LIN {X 0,Y 485.77,Z 296.531,A -85,B 0,C 180,E1 -14643.447,E2 -14643.447} C_VEL
LIN {X 0,Y 485.784,Z 296.534,A -85,B 0,C 180,E1 -14646.187,E2 -14646.187} C_VEL
LIN {X 0,Y 485.815,Z 296.524,A -85,B 0,C 180,E1 -14648.87,E2 -14648.87} C_VEL
LIN {X 0,Y 485.863,Z 296.525,A -85,B 0,C 180,E1 -14652.08,E2 -14652.08} C_VEL
LIN {X 0,Y 485.883,Z 296.515,A -85,B 0,C 180,E1 -14654.987,E2 -14654.987} C_VEL
LIN {X 0,Y 485.919,Z 296.513,A -85,B 0,C 180,E1 -14658.355,E2 -14658.355} C_VEL
LIN {X 0,Y 485.937,Z 296.624,A -85,B 0,C 180,E1 -14661.371,E2 -14661.371} C_VEL
LIN {X 0,Y 487.362,Z 304.386,A -85,B 0,C 180,E1 -14663.005,E2 -14663.005} C_VEL
LIN {X 0,Y 489.641,Z 313.003,A -85,B 0,C 180,E1 -14663.215,E2 -14663.215} C_VEL
LIN {X 0,Y 492.442,Z 326.863,A -85,B 0,C 180,E1 -14663.515,E2 -14663.515} C_VEL
LIN {X 0,Y 490.89,Z 439.426,A -85,B 0,C 180,E1 -14665.164,E2 -14665.164} C_VEL
LIN {X 0,Y 490.643,Z 451.445,A -85,B 0,C 180,E1 -14665.464,E2 -14665.464} C_VEL
LIN {X 0,Y 489.693,Z 457.148,A -85,B 0,C 180,E1 -14665.617,E2 -14665.617} C_VEL
LIN {X 0,Y 486.571,Z 466.299,A -85,B 0,C 180,E1 -14665.884,E2 -14665.884} C_VEL
LIN {X 0,Y 483.496,Z 475.212,A -85,B 0,C 180,E1 -14666.236,E2 -14666.236} C_VEL
LIN {X 0,Y 482.618,Z 480.534,A -85,B 0,C 180,E1 -14666.517,E2 -14666.517} C_VEL
LIN {X 0,Y 481.935,Z 493.871,A -85,B 0,C 180,E1 -14667.395,E2 -14667.395} C_VEL
LIN {X 0,Y 480.98,Z 505.372,A -85,B 0,C 180,E1 -14668.329,E2 -14668.329} C_VEL
LIN {X 0,Y 480.395,Z 515.838,A -85,B 0,C 180,E1 -14669.371,E2 -14669.371} C_VEL
LIN {X 0,Y 479.518,Z 526.296,A -85,B 0,C 180,E1 -14670.626,E2 -14670.626} C_VEL
LIN {X 0,Y 478.886,Z 534.915,A -85,B 0,C 180,E1 -14671.884,E2 -14671.884} C_VEL
LIN {X 0,Y 478.287,Z 542.104,A -85,B 0,C 180,E1 -14673.146,E2 -14673.146} C_VEL
LIN {X 0,Y 477.979,Z 549.726,A -85,B 0,C 180,E1 -14674.801,E2 -14674.801} C_VEL
LIN {X 0,Y 477.604,Z 555.152,A -85,B 0,C 180,E1 -14676.313,E2 -14676.313} C_VEL
LIN {X 0,Y 477.361,Z 558.684,A -85,B 0,C 180,E1 -14677.586,E2 -14677.586} C_VEL
LIN {X 0,Y 477.178,Z 562.146,A -85,B 0,C 180,E1 -14679.29,E2 -14679.29} C_VEL
LIN {X 0,Y 477.117,Z 564.216,A -85,B 0,C 180,E1 -14681,E2 -14681} C_VEL
LIN {X 0,Y 477.101,Z 564.93,A -85,B 0,C 180,E1 -14682.72,E2 -14682.72} C_VEL
LIN {X 0,Y 477.337,Z 564.263,A -85,B 0,C 180,E1 -14684.443,E2 -14684.443} C_VEL
LIN {X 0,Y 477.485,Z 562.216,A -85,B 0,C 180,E1 -14686.181,E2 -14686.181} C_VEL
LIN {X 0,Y 477.942,Z 558.707,A -85,B 0,C 180,E1 -14687.922,E2 -14687.922} C_VEL
LIN {X 0,Y 478.56,Z 553.62,A -85,B 0,C 180,E1 -14689.67,E2 -14689.67} C_VEL
LIN {X 0,Y 479.118,Z 548.633,A -85,B 0,C 180,E1 -14690.985,E2 -14690.985} C_VEL
LIN {X 0,Y 480.003,Z 541.388,A -85,B 0,C 180,E1 -14692.52,E2 -14692.52} C_VEL
LIN {X 0,Y 480.959,Z 533.698,A -85,B 0,C 180,E1 -14693.839,E2 -14693.839} C_VEL
LIN {X 0,Y 482.026,Z 524.437,A -85,B 0,C 180,E1 -14695.15,E2 -14695.15} C_VEL
LIN {X 0,Y 483.19,Z 514.097,A -85,B 0,C 180,E1 -14696.353,E2 -14696.353} C_VEL
LIN {X 0,Y 484.363,Z 502.622,A -85,B 0,C 180,E1 -14697.446,E2 -14697.446} C_VEL
LIN {X 0,Y 485.333,Z 491.49,A -85,B 0,C 180,E1 -14698.313,E2 -14698.313} C_VEL
LIN {X 0,Y 486.333,Z 478.223,A -85,B 0,C 180,E1 -14699.14,E2 -14699.14} C_VEL
LIN {X 0,Y 487.079,Z 464.484,A -85,B 0,C 180,E1 -14699.801,E2 -14699.801} C_VEL
LIN {X 0,Y 487.718,Z 449.719,A -85,B 0,C 180,E1 -14700.31,E2 -14700.31} C_VEL
LIN {X 0,Y 488.109,Z 435.76,A -85,B 0,C 180,E1 -14700.619,E2 -14700.619} C_VEL
LIN {X 0,Y 489.875,Z 330.426,A -85,B 0,C 180,E1 -14702.194,E2 -14702.194} C_VEL
LIN {X 0,Y 488.073,Z 324.325,A -85,B 0,C 180,E1 -14702.385,E2 -14702.385} C_VEL
LIN {X 0,Y 480.502,Z 305.747,A -85,B 0,C 180,E1 -14703.112,E2 -14703.112} C_VEL
LIN {X 0,Y 478.693,Z 297.414,A -85,B 0,C 180,E1 -14705.071,E2 -14705.071} C_VEL
LIN {X 0,Y 478.681,Z 297.417,A -85,B 0,C 180,E1 -14707.918,E2 -14707.918} C_VEL
LIN {X 0,Y 478.695,Z 297.409,A -85,B 0,C 180,E1 -14711.179,E2 -14711.179} C_VEL
LIN {X 0,Y 478.716,Z 297.403,A -85,B 0,C 180,E1 -14714.196,E2 -14714.196} C_VEL
LIN {X 0,Y 478.703,Z 297.412,A -85,B 0,C 180,E1 -14717.017,E2 -14717.017} C_VEL
LIN {X 0,Y 478.708,Z 297.412,A -85,B 0,C 180,E1 -14719.924,E2 -14719.924} C_VEL
LIN {X 0,Y 478.721,Z 297.402,A -85,B 0,C 180,E1 -14723.138,E2 -14723.138} C_VEL
LIN {X 0,Y 478.69,Z 297.412,A -85,B 0,C 180,E1 -14726.218,E2 -14726.218} C_VEL
LIN {X 0,Y 478.703,Z 297.407,A -85,B 0,C 180,E1 -14729.195,E2 -14729.195} C_VEL
LIN {X 0,Y 478.741,Z 297.401,A -85,B 0,C 180,E1 -14732.083,E2 -14732.083} C_VEL
LIN {X 0,Y 478.725,Z 297.41,A -85,B 0,C 180,E1 -14735.108,E2 -14735.108} C_VEL
LIN {X 0,Y 478.751,Z 297.404,A -85,B 0,C 180,E1 -14738.545,E2 -14738.545} C_VEL
LIN {X 0,Y 478.762,Z 297.398,A -85,B 0,C 180,E1 -14741.224,E2 -14741.224} C_VEL
LIN {X 0,Y 478.812,Z 297.397,A -85,B 0,C 180,E1 -14744.895,E2 -14744.895} C_VEL
LIN {X 0,Y 478.849,Z 297.392,A -85,B 0,C 180,E1 -14748.183,E2 -14748.183} C_VEL
LIN {X 0,Y 478.887,Z 297.383,A -85,B 0,C 180,E1 -14751.589,E2 -14751.589} C_VEL
LIN {X 0,Y 478.991,Z 297.376,A -85,B 0,C 180,E1 -14754.966,E2 -14754.966} C_VEL
LIN {X 0,Y 478.798,Z 297.397,A -85,B 0,C 180,E1 -14757.485,E2 -14757.485} C_VEL
LIN {X 0,Y 479.032,Z 297.368,A -85,B 0,C 180,E1 -14760,E2 -14760} C_VEL
LIN {X 0,Y 478.98,Z 297.375,A -85,B 0,C 180,E1 -14764.193,E2 -14764.193} C_VEL
LIN {X 0,Y 478.917,Z 297.378,A -85,B 0,C 180,E1 -14766.719,E2 -14766.719} C_VEL
LIN {X 0,Y 478.863,Z 297.392,A -85,B 0,C 180,E1 -14769.259,E2 -14769.259} C_VEL
LIN {X 0,Y 478.898,Z 297.377,A -85,B 0,C 180,E1 -14771.816,E2 -14771.816} C_VEL
LIN {X 0,Y 478.856,Z 297.39,A -85,B 0,C 180,E1 -14775.266,E2 -14775.266} C_VEL
LIN {X 0,Y 478.778,Z 297.398,A -85,B 0,C 180,E1 -14778.775,E2 -14778.775} C_VEL
LIN {X 0,Y 478.751,Z 297.397,A -85,B 0,C 180,E1 -14781.455,E2 -14781.455} C_VEL
LIN {X 0,Y 478.725,Z 297.409,A -85,B 0,C 180,E1 -14784.892,E2 -14784.892} C_VEL
LIN {X 0,Y 478.741,Z 297.405,A -85,B 0,C 180,E1 -14787.917,E2 -14787.917} C_VEL
LIN {X 0,Y 478.725,Z 297.407,A -85,B 0,C 180,E1 -14790.804,E2 -14790.804} C_VEL
LIN {X 0,Y 478.741,Z 297.404,A -85,B 0,C 180,E1 -14793.778,E2 -14793.778} C_VEL
LIN {X 0,Y 478.784,Z 297.387,A -85,B 0,C 180,E1 -14796.857,E2 -14796.857} C_VEL
LIN {X 0,Y 478.754,Z 297.405,A -85,B 0,C 180,E1 -14800.072,E2 -14800.072} C_VEL
LIN {X 0,Y 478.732,Z 297.406,A -85,B 0,C 180,E1 -14803.446,E2 -14803.446} C_VEL
LIN {X 0,Y 478.719,Z 297.411,A -85,B 0,C 180,E1 -14806.556,E2 -14806.556} C_VEL
LIN {X 0,Y 478.747,Z 297.406,A -85,B 0,C 180,E1 -14809.535,E2 -14809.535} C_VEL
LIN {X 0,Y 478.781,Z 297.408,A -85,B 0,C 180,E1 -14812.186,E2 -14812.186} C_VEL
LIN {X 0,Y 478.744,Z 297.414,A -85,B 0,C 180,E1 -14815.211,E2 -14815.211} C_VEL
LIN {X 0,Y 478.763,Z 297.414,A -85,B 0,C 180,E1 -14818.221,E2 -14818.221} C_VEL
LIN {X 0,Y 478.75,Z 297.508,A -85,B 0,C 180,E1 -14819.048,E2 -14819.048} C_VEL
LIN {X 0,Y 482.247,Z 312.121,A -85,B 0,C 180,E1 -14821.836,E2 -14821.836} C_VEL
LIN {X 0,Y 484.81,Z 324.657,A -85,B 0,C 180,E1 -14824.101,E2 -14824.101} C_VEL
LIN {X 0,Y 483.591,Z 338.406,A -85,B 0,C 180,E1 -14826.303,E2 -14826.303} C_VEL
LIN {X 0,Y 481.96,Z 355.754,A -85,B 0,C 180,E1 -14829.033,E2 -14829.033} C_VEL
LIN {X 0,Y 486.987,Z 384.746,A -85,B 0,C 180,E1 -14829.76,E2 -14829.76} C_VEL
LIN {X 0,Y 488.865,Z 398.674,A -85,B 0,C 180,E1 -14830.074,E2 -14830.074} C_VEL
LIN {X 0,Y 487.289,Z 493.967,A -85,B 0,C 180,E1 -14831.513,E2 -14831.513} C_VEL
LIN {X 0,Y 486.53,Z 508.818,A -85,B 0,C 180,E1 -14831.899,E2 -14831.899} C_VEL
LIN {X 0,Y 485.571,Z 522.508,A -85,B 0,C 180,E1 -14832.423,E2 -14832.423} C_VEL
LIN {X 0,Y 484.462,Z 535.489,A -85,B 0,C 180,E1 -14833.086,E2 -14833.086} C_VEL
LIN {X 0,Y 483.26,Z 548.083,A -85,B 0,C 180,E1 -14833.909,E2 -14833.909} C_VEL
LIN {X 0,Y 481.995,Z 559.586,A -85,B 0,C 180,E1 -14834.839,E2 -14834.839} C_VEL
LIN {X 0,Y 480.873,Z 570.17,A -85,B 0,C 180,E1 -14835.881,E2 -14835.881} C_VEL
LIN {X 0,Y 479.709,Z 580.705,A -85,B 0,C 180,E1 -14837.136,E2 -14837.136} C_VEL
LIN {X 0,Y 478.789,Z 590.546,A -85,B 0,C 180,E1 -14838.573,E2 -14838.573} C_VEL
LIN {X 0,Y 477.939,Z 598.91,A -85,B 0,C 180,E1 -14840.086,E2 -14840.086} C_VEL
LIN {X 0,Y 477.375,Z 605.499,A -85,B 0,C 180,E1 -14841.565,E2 -14841.565} C_VEL
LIN {X 0,Y 476.995,Z 617.328,A -85,B 0,C 180,E1 -14844.947,E2 -14844.947} C_VEL
LIN {X 0,Y 476.94,Z 621.761,A -85,B 0,C 180,E1 -14846.634,E2 -14846.634} C_VEL
LIN {X 0,Y 476.957,Z 624.638,A -85,B 0,C 180,E1 -14848.319,E2 -14848.319} C_VEL
LIN {X 0,Y 477.003,Z 625.52,A -85,B 0,C 180,E1 -14849.161,E2 -14849.161} C_VEL
LIN {X 0,Y 476.959,Z 626.175,A -85,B 0,C 180,E1 -14850.843,E2 -14850.843} C_VEL
LIN {X 0,Y 476.924,Z 625.353,A -85,B 0,C 180,E1 -14852.527,E2 -14852.527} C_VEL
LIN {X 0,Y 476.963,Z 623.088,A -85,B 0,C 180,E1 -14854.213,E2 -14854.213} C_VEL
LIN {X 0,Y 477.08,Z 619.333,A -85,B 0,C 180,E1 -14855.901,E2 -14855.901} C_VEL
LIN {X 0,Y 477.383,Z 614.001,A -85,B 0,C 180,E1 -14857.59,E2 -14857.59} C_VEL
LIN {X 0,Y 477.739,Z 608.828,A -85,B 0,C 180,E1 -14858.858,E2 -14858.858} C_VEL
LIN {X 0,Y 478.476,Z 601.406,A -85,B 0,C 180,E1 -14860.333,E2 -14860.333} C_VEL
LIN {X 0,Y 479.204,Z 593.155,A -85,B 0,C 180,E1 -14861.67,E2 -14861.67} C_VEL
LIN {X 0,Y 480.028,Z 584.334,A -85,B 0,C 180,E1 -14862.859,E2 -14862.859} C_VEL
LIN {X 0,Y 480.975,Z 574.091,A -85,B 0,C 180,E1 -14864.013,E2 -14864.013} C_VEL
LIN {X 0,Y 482.133,Z 562.839,A -85,B 0,C 180,E1 -14865.053,E2 -14865.053} C_VEL
LIN {X 0,Y 483.157,Z 550.55,A -85,B 0,C 180,E1 -14865.991,E2 -14865.991} C_VEL
LIN {X 0,Y 484.352,Z 536.947,A -85,B 0,C 180,E1 -14866.814,E2 -14866.814} C_VEL
LIN {X 0,Y 485.362,Z 522.74,A -85,B 0,C 180,E1 -14867.481,E2 -14867.481} C_VEL
LIN {X 0,Y 486.254,Z 508.664,A -85,B 0,C 180,E1 -14867.959,E2 -14867.959} C_VEL
LIN {X 0,Y 486.975,Z 491.209,A -85,B 0,C 180,E1 -14868.346,E2 -14868.346} C_VEL
LIN {X 0,Y 489.953,Z 399.064,A -85,B 0,C 180,E1 -14870.171,E2 -14870.171} C_VEL
LIN {X 0,Y 488.283,Z 381.463,A -85,B 0,C 180,E1 -14870.68,E2 -14870.68} C_VEL
LIN {X 0,Y 484.759,Z 358.037,A -85,B 0,C 180,E1 -14871.468,E2 -14871.468} C_VEL
LIN {X 0,Y 483.933,Z 352.73,A -85,B 0,C 180,E1 -14871.699,E2 -14871.699} C_VEL
LIN {X 0,Y 481.685,Z 333.484,A -85,B 0,C 180,E1 -14872.865,E2 -14872.865} C_VEL
LIN {X 0,Y 482.771,Z 318.818,A -85,B 0,C 180,E1 -14875.113,E2 -14875.113} C_VEL
LIN {X 0,Y 480.649,Z 306.868,A -85,B 0,C 180,E1 -14877.094,E2 -14877.094} C_VEL
LIN {X 0,Y 478.775,Z 297.404,A -85,B 0,C 180,E1 -14878.705,E2 -14878.705} C_VEL
LIN {X 0,Y 478.675,Z 297.414,A -85,B 0,C 180,E1 -14881.928,E2 -14881.928} C_VEL
LIN {X 0,Y 478.711,Z 297.414,A -85,B 0,C 180,E1 -14884.977,E2 -14884.977} C_VEL
LIN {X 0,Y 478.676,Z 297.417,A -85,B 0,C 180,E1 -14887.924,E2 -14887.924} C_VEL
LIN {X 0,Y 478.708,Z 297.412,A -85,B 0,C 180,E1 -14890.46,E2 -14890.46} C_VEL
LIN {X 0,Y 478.739,Z 297.408,A -85,B 0,C 180,E1 -14893.447,E2 -14893.447} C_VEL
LIN {X 0,Y 478.74,Z 297.409,A -85,B 0,C 180,E1 -14896.555,E2 -14896.555} C_VEL
LIN {X 0,Y 478.708,Z 297.411,A -85,B 0,C 180,E1 -14899.542,E2 -14899.542} C_VEL
LIN {X 0,Y 478.71,Z 297.413,A -85,B 0,C 180,E1 -14902.199,E2 -14902.199} C_VEL
LIN {X 0,Y 478.747,Z 297.408,A -85,B 0,C 180,E1 -14905.208,E2 -14905.208} C_VEL
LIN {X 0,Y 478.718,Z 297.413,A -85,B 0,C 180,E1 -14908.214,E2 -14908.214} C_VEL
LIN {X 0,Y 478.757,Z 297.405,A -85,B 0,C 180,E1 -14911.384,E2 -14911.384} C_VEL
LIN {X 0,Y 478.733,Z 297.412,A -85,B 0,C 180,E1 -14913.964,E2 -14913.964} C_VEL
LIN {X 0,Y 478.761,Z 297.411,A -85,B 0,C 180,E1 -14917.181,E2 -14917.181} C_VEL
LIN {X 0,Y 478.785,Z 297.414,A -85,B 0,C 180,E1 -14920.337,E2 -14920.337} C_VEL
LIN {X 0,Y 478.83,Z 297.543,A -85,B 0,C 180,E1 -14922.632,E2 -14922.632} C_VEL
LIN {X 0,Y 483.17,Z 311.983,A -85,B 0,C 180,E1 -14925.304,E2 -14925.304} C_VEL
LIN {X 0,Y 486.011,Z 325.005,A -85,B 0,C 180,E1 -14927.515,E2 -14927.515} C_VEL
LIN {X 0,Y 486.185,Z 329.106,A -85,B 0,C 180,E1 -14928.153,E2 -14928.153} C_VEL
LIN {X 0,Y 485.162,Z 345.213,A -85,B 0,C 180,E1 -14930.495,E2 -14930.495} C_VEL
LIN {X 0,Y 490.051,Z 367.792,A -85,B 0,C 180,E1 -14931.354,E2 -14931.354} C_VEL
LIN {X 0,Y 491.129,Z 374.172,A -85,B 0,C 180,E1 -14931.568,E2 -14931.568} C_VEL
LIN {X 0,Y 487.703,Z 474.381,A -85,B 0,C 180,E1 -14933.532,E2 -14933.532} C_VEL
LIN {X 0,Y 487.049,Z 490.57,A -85,B 0,C 180,E1 -14933.912,E2 -14933.912} C_VEL
LIN {X 0,Y 486.356,Z 504.272,A -85,B 0,C 180,E1 -14934.396,E2 -14934.396} C_VEL
LIN {X 0,Y 485.275,Z 518.802,A -85,B 0,C 180,E1 -14935.083,E2 -14935.083} C_VEL
LIN {X 0,Y 484.276,Z 531.323,A -85,B 0,C 180,E1 -14935.853,E2 -14935.853} C_VEL
LIN {X 0,Y 483.13,Z 543.526,A -85,B 0,C 180,E1 -14936.779,E2 -14936.779} C_VEL
LIN {X 0,Y 482.019,Z 555.678,A -85,B 0,C 180,E1 -14937.918,E2 -14937.918} C_VEL
LIN {X 0,Y 480.878,Z 566.583,A -85,B 0,C 180,E1 -14939.165,E2 -14939.165} C_VEL
LIN {X 0,Y 479.753,Z 575.623,A -85,B 0,C 180,E1 -14940.418,E2 -14940.418} C_VEL
LIN {X 0,Y 478.88,Z 584.231,A -85,B 0,C 180,E1 -14941.886,E2 -14941.886} C_VEL
LIN {X 0,Y 478.087,Z 591.225,A -85,B 0,C 180,E1 -14943.36,E2 -14943.36} C_VEL
LIN {X 0,Y 477.836,Z 595.873,A -85,B 0,C 180,E1 -14944.579,E2 -14944.579} C_VEL
LIN {X 0,Y 477.453,Z 599.934,A -85,B 0,C 180,E1 -14945.894,E2 -14945.894} C_VEL
LIN {X 0,Y 477.069,Z 603.711,A -85,B 0,C 180,E1 -14947.593,E2 -14947.593} C_VEL
LIN {X 0,Y 476.906,Z 606.01,A -85,B 0,C 180,E1 -14949.297,E2 -14949.297} C_VEL
LIN {X 0,Y 476.914,Z 606.669,A -85,B 0,C 180,E1 -14950.247,E2 -14950.247} C_VEL
LIN {X 0,Y 476.739,Z 606.749,A -85,B 0,C 180,E1 -14951.87,E2 -14951.87} C_VEL
LIN {X 0,Y 476.784,Z 605.387,A -85,B 0,C 180,E1 -14953.595,E2 -14953.595} C_VEL
LIN {X 0,Y 476.834,Z 604.117,A -85,B 0,C 180,E1 -14954.461,E2 -14954.461} C_VEL
LIN {X 0,Y 476.931,Z 600.386,A -85,B 0,C 180,E1 -14956.203,E2 -14956.203} C_VEL
LIN {X 0,Y 477.083,Z 596.142,A -85,B 0,C 180,E1 -14957.614,E2 -14957.614} C_VEL
LIN {X 0,Y 477.386,Z 589.572,A -85,B 0,C 180,E1 -14959.277,E2 -14959.277} C_VEL
LIN {X 0,Y 477.755,Z 581.739,A -85,B 0,C 180,E1 -14960.826,E2 -14960.826} C_VEL
LIN {X 0,Y 478.214,Z 573.386,A -85,B 0,C 180,E1 -14962.158,E2 -14962.158} C_VEL
LIN {X 0,Y 478.832,Z 563.194,A -85,B 0,C 180,E1 -14963.492,E2 -14963.492} C_VEL
LIN {X 0,Y 479.486,Z 551.781,A -85,B 0,C 180,E1 -14964.719,E2 -14964.719} C_VEL
LIN {X 0,Y 480.154,Z 540.357,A -85,B 0,C 180,E1 -14965.727,E2 -14965.727} C_VEL
LIN {X 0,Y 480.828,Z 528.102,A -85,B 0,C 180,E1 -14966.612,E2 -14966.612} C_VEL
LIN {X 0,Y 481.466,Z 514.839,A -85,B 0,C 180,E1 -14967.377,E2 -14967.377} C_VEL
LIN {X 0,Y 482.085,Z 500.781,A -85,B 0,C 180,E1 -14968.001,E2 -14968.001} C_VEL
LIN {X 0,Y 482.647,Z 486.247,A -85,B 0,C 180,E1 -14968.467,E2 -14968.467} C_VEL
LIN {X 0,Y 483.012,Z 468.488,A -85,B 0,C 180,E1 -14968.828,E2 -14968.828} C_VEL
LIN {X 0,Y 484.847,Z 370.517,A -85,B 0,C 180,E1 -14970.589,E2 -14970.589} C_VEL
LIN {X 0,Y 481.086,Z 343.578,A -85,B 0,C 180,E1 -14971.22,E2 -14971.22} C_VEL
LIN {X 0,Y 481.95,Z 323.747,A -85,B 0,C 180,E1 -14974.062,E2 -14974.062} C_VEL
LIN {X 0,Y 482.272,Z 315.444,A -85,B 0,C 180,E1 -14975.255,E2 -14975.255} C_VEL
LIN {X 0,Y 479,Z 298.562,A -85,B 0,C 180,E1 -14977.846,E2 -14977.846} C_VEL
LIN {X 0,Y 478.724,Z 297.412,A -85,B 0,C 180,E1 -14978.05,E2 -14978.05} C_VEL
LIN {X 0,Y 478.719,Z 297.408,A -85,B 0,C 180,E1 -14981.18,E2 -14981.18} C_VEL
LIN {X 0,Y 478.739,Z 297.411,A -85,B 0,C 180,E1 -14984.197,E2 -14984.197} C_VEL
LIN {X 0,Y 478.714,Z 297.409,A -85,B 0,C 180,E1 -14987.02,E2 -14987.02} C_VEL
LIN {X 0,Y 478.696,Z 297.414,A -85,B 0,C 180,E1 -14989.921,E2 -14989.921} C_VEL
LIN {X 0,Y 478.674,Z 297.414,A -85,B 0,C 180,E1 -14993.132,E2 -14993.132} C_VEL
LIN {X 0,Y 478.701,Z 297.416,A -85,B 0,C 180,E1 -14996.217,E2 -14996.217} C_VEL
LIN {X 0,Y 478.723,Z 297.41,A -85,B 0,C 180,E1 -14999.685,E2 -14999.685} C_VEL
LIN {X 0,Y 478.743,Z 297.411,A -85,B 0,C 180,E1 -15002.081,E2 -15002.081} C_VEL
LIN {X 0,Y 478.752,Z 297.404,A -85,B 0,C 180,E1 -15005.108,E2 -15005.108} C_VEL
LIN {X 0,Y 478.78,Z 297.402,A -85,B 0,C 180,E1 -15008.545,E2 -15008.545} C_VEL
LIN {X 0,Y 478.824,Z 297.401,A -85,B 0,C 180,E1 -15011.961,E2 -15011.961} C_VEL
LIN {X 0,Y 478.843,Z 297.392,A -85,B 0,C 180,E1 -15014.892,E2 -15014.892} C_VEL
LIN {X 0,Y 478.876,Z 297.392,A -85,B 0,C 180,E1 -15018.182,E2 -15018.182} C_VEL
LIN {X 0,Y 478.9,Z 297.528,A -85,B 0,C 180,E1 -15021.217,E2 -15021.217} C_VEL
LIN {X 0,Y 480.268,Z 304.765,A -85,B 0,C 180,E1 -15022.76,E2 -15022.76} C_VEL
LIN {X 0,Y 482.973,Z 314.716,A -85,B 0,C 180,E1 -15023.016,E2 -15023.016} C_VEL
LIN {X 0,Y 485.65,Z 329.013,A -85,B 0,C 180,E1 -15023.323,E2 -15023.323} C_VEL
LIN {X 0,Y 484.007,Z 439.783,A -85,B 0,C 180,E1 -15024.965,E2 -15024.965} C_VEL
LIN {X 0,Y 483.662,Z 454.476,A -85,B 0,C 180,E1 -15025.351,E2 -15025.351} C_VEL
LIN {X 0,Y 483.145,Z 468.419,A -85,B 0,C 180,E1 -15025.893,E2 -15025.893} C_VEL
LIN {X 0,Y 482.618,Z 480.534,A -85,B 0,C 180,E1 -15026.517,E2 -15026.517} C_VEL
LIN {X 0,Y 481.676,Z 485.877,A -85,B 0,C 180,E1 -15026.822,E2 -15026.822} C_VEL
LIN {X 0,Y 478.298,Z 494.251,A -85,B 0,C 180,E1 -15027.321,E2 -15027.321} C_VEL
LIN {X 0,Y 474.914,Z 502.288,A -85,B 0,C 180,E1 -15027.879,E2 -15027.879} C_VEL
LIN {X 0,Y 473.928,Z 506.979,A -85,B 0,C 180,E1 -15028.284,E2 -15028.284} C_VEL
LIN {X 0,Y 473.357,Z 517.422,A -85,B 0,C 180,E1 -15029.362,E2 -15029.362} C_VEL
LIN {X 0,Y 472.427,Z 527.691,A -85,B 0,C 180,E1 -15030.635,E2 -15030.635} C_VEL
LIN {X 0,Y 471.824,Z 536.145,A -85,B 0,C 180,E1 -15031.912,E2 -15031.912} C_VEL
LIN {X 0,Y 471.114,Z 544.258,A -85,B 0,C 180,E1 -15033.407,E2 -15033.407} C_VEL
LIN {X 0,Y 470.913,Z 550.161,A -85,B 0,C 180,E1 -15034.746,E2 -15034.746} C_VEL
LIN {X 0,Y 470.499,Z 555.958,A -85,B 0,C 180,E1 -15036.409,E2 -15036.409} C_VEL
LIN {X 0,Y 470.245,Z 559.431,A -85,B 0,C 180,E1 -15037.702,E2 -15037.702} C_VEL
LIN {X 0,Y 470.084,Z 562.787,A -85,B 0,C 180,E1 -15039.431,E2 -15039.431} C_VEL
LIN {X 0,Y 470.029,Z 564.736,A -85,B 0,C 180,E1 -15041.168,E2 -15041.168} C_VEL
LIN {X 0,Y 470.034,Z 565.327,A -85,B 0,C 180,E1 -15042.914,E2 -15042.914} C_VEL
LIN {X 0,Y 470.265,Z 564.557,A -85,B 0,C 180,E1 -15044.665,E2 -15044.665} C_VEL
LIN {X 0,Y 470.457,Z 562.408,A -85,B 0,C 180,E1 -15046.43,E2 -15046.43} C_VEL
LIN {X 0,Y 470.959,Z 558.794,A -85,B 0,C 180,E1 -15048.197,E2 -15048.197} C_VEL
LIN {X 0,Y 471.637,Z 553.596,A -85,B 0,C 180,E1 -15049.971,E2 -15049.971} C_VEL
LIN {X 0,Y 472.229,Z 548.487,A -85,B 0,C 180,E1 -15051.307,E2 -15051.307} C_VEL
LIN {X 0,Y 473.183,Z 541.11,A -85,B 0,C 180,E1 -15052.863,E2 -15052.863} C_VEL
LIN {X 0,Y 474.19,Z 533.298,A -85,B 0,C 180,E1 -15054.196,E2 -15054.196} C_VEL
LIN {X 0,Y 475.335,Z 523.936,A -85,B 0,C 180,E1 -15055.516,E2 -15055.516} C_VEL
LIN {X 0,Y 476.56,Z 513.234,A -85,B 0,C 180,E1 -15056.749,E2 -15056.749} C_VEL
LIN {X 0,Y 477.822,Z 501.422,A -85,B 0,C 180,E1 -15057.854,E2 -15057.854} C_VEL
LIN {X 0,Y 478.829,Z 490.016,A -85,B 0,C 180,E1 -15058.727,E2 -15058.727} C_VEL
LIN {X 0,Y 479.822,Z 477.164,A -85,B 0,C 180,E1 -15059.514,E2 -15059.514} C_VEL
LIN {X 0,Y 480.516,Z 464.313,A -85,B 0,C 180,E1 -15060.129,E2 -15060.129} C_VEL
LIN {X 0,Y 481.157,Z 449.886,A -85,B 0,C 180,E1 -15060.628,E2 -15060.628} C_VEL
LIN {X 0,Y 481.555,Z 436.381,A -85,B 0,C 180,E1 -15060.93,E2 -15060.93} C_VEL
LIN {X 0,Y 483.353,Z 331.59,A -85,B 0,C 180,E1 -15062.519,E2 -15062.519} C_VEL
LIN {X 0,Y 481.848,Z 326.725,A -85,B 0,C 180,E1 -15062.679,E2 -15062.679} C_VEL
LIN {X 0,Y 474.63,Z 309.241,A -85,B 0,C 180,E1 -15063.368,E2 -15063.368} C_VEL
LIN {X 0,Y 473.384,Z 306.242,A -85,B 0,C 180,E1 -15063.503,E2 -15063.503} C_VEL
LIN {X 0,Y 471.633,Z 298.296,A -85,B 0,C 180,E1 -15065.424,E2 -15065.424} C_VEL
LIN {X 0,Y 471.621,Z 298.29,A -85,B 0,C 180,E1 -15068.589,E2 -15068.589} C_VEL
LIN {X 0,Y 471.653,Z 298.286,A -85,B 0,C 180,E1 -15071.931,E2 -15071.931} C_VEL
LIN {X 0,Y 471.69,Z 298.274,A -85,B 0,C 180,E1 -15074.538,E2 -15074.538} C_VEL
LIN {X 0,Y 471.653,Z 298.291,A -85,B 0,C 180,E1 -15077.944,E2 -15077.944} C_VEL
LIN {X 0,Y 471.671,Z 298.288,A -85,B 0,C 180,E1 -15080.549,E2 -15080.549} C_VEL
LIN {X 0,Y 471.685,Z 298.27,A -85,B 0,C 180,E1 -15083.559,E2 -15083.559} C_VEL
LIN {X 0,Y 471.639,Z 298.29,A -85,B 0,C 180,E1 -15086.667,E2 -15086.667} C_VEL
LIN {X 0,Y 471.679,Z 298.285,A -85,B 0,C 180,E1 -15089.675,E2 -15089.675} C_VEL
LIN {X 0,Y 471.704,Z 298.275,A -85,B 0,C 180,E1 -15092.987,E2 -15092.987} C_VEL
LIN {X 0,Y 471.666,Z 298.291,A -85,B 0,C 180,E1 -15095.43,E2 -15095.43} C_VEL
LIN {X 0,Y 471.708,Z 298.283,A -85,B 0,C 180,E1 -15098.209,E2 -15098.209} C_VEL
LIN {X 0,Y 471.704,Z 298.277,A -85,B 0,C 180,E1 -15100.932,E2 -15100.932} C_VEL
LIN {X 0,Y 471.736,Z 298.277,A -85,B 0,C 180,E1 -15104.498,E2 -15104.498} C_VEL
LIN {X 0,Y 471.768,Z 298.27,A -85,B 0,C 180,E1 -15107.132,E2 -15107.132} C_VEL
LIN {X 0,Y 471.785,Z 298.268,A -85,B 0,C 180,E1 -15109.737,E2 -15109.737} C_VEL
LIN {X 0,Y 471.865,Z 298.258,A -85,B 0,C 180,E1 -15112.322,E2 -15112.322} C_VEL
LIN {X 0,Y 471.938,Z 298.256,A -85,B 0,C 180,E1 -15114.891,E2 -15114.891} C_VEL
LIN {X 0,Y 471.772,Z 298.272,A -85,B 0,C 180,E1 -15117.447,E2 -15117.447} C_VEL
LIN {X 0,Y 471.986,Z 298.245,A -85,B 0,C 180,E1 -15120,E2 -15120} C_VEL
LIN {X 0,Y 471.948,Z 298.251,A -85,B 0,C 180,E1 -15124.256,E2 -15124.256} C_VEL
LIN {X 0,Y 471.869,Z 298.254,A -85,B 0,C 180,E1 -15126.82,E2 -15126.82} C_VEL
LIN {X 0,Y 471.828,Z 298.267,A -85,B 0,C 180,E1 -15129.398,E2 -15129.398} C_VEL
LIN {X 0,Y 471.857,Z 298.254,A -85,B 0,C 180,E1 -15131.995,E2 -15131.995} C_VEL
LIN {X 0,Y 471.78,Z 298.27,A -85,B 0,C 180,E1 -15135.5,E2 -15135.5} C_VEL
LIN {X 0,Y 471.759,Z 298.265,A -85,B 0,C 180,E1 -15138.168,E2 -15138.168} C_VEL
LIN {X 0,Y 471.707,Z 298.28,A -85,B 0,C 180,E1 -15140.878,E2 -15140.878} C_VEL
LIN {X 0,Y 471.655,Z 298.286,A -85,B 0,C 180,E1 -15143.639,E2 -15143.639} C_VEL
LIN {X 0,Y 471.679,Z 298.282,A -85,B 0,C 180,E1 -15146.455,E2 -15146.455} C_VEL
LIN {X 0,Y 471.678,Z 298.284,A -85,B 0,C 180,E1 -15149.344,E2 -15149.344} C_VEL
LIN {X 0,Y 471.686,Z 298.289,A -85,B 0,C 180,E1 -15152.316,E2 -15152.316} C_VEL
LIN {X 0,Y 471.707,Z 298.257,A -85,B 0,C 180,E1 -15155.388,E2 -15155.388} C_VEL
LIN {X 0,Y 471.709,Z 298.28,A -85,B 0,C 180,E1 -15158.098,E2 -15158.098} C_VEL
LIN {X 0,Y 471.687,Z 298.287,A -85,B 0,C 180,E1 -15160.798,E2 -15160.798} C_VEL
LIN {X 0,Y 471.686,Z 298.29,A -85,B 0,C 180,E1 -15164.262,E2 -15164.262} C_VEL
LIN {X 0,Y 471.679,Z 298.285,A -85,B 0,C 180,E1 -15166.917,E2 -15166.917} C_VEL
LIN {X 0,Y 471.718,Z 298.287,A -85,B 0,C 180,E1 -15170.324,E2 -15170.324} C_VEL
LIN {X 0,Y 471.745,Z 298.274,A -85,B 0,C 180,E1 -15173.568,E2 -15173.568} C_VEL
LIN {X 0,Y 471.687,Z 298.287,A -85,B 0,C 180,E1 -15176.674,E2 -15176.674} C_VEL
LIN {X 0,Y 471.716,Z 298.385,A -85,B 0,C 180,E1 -15178.69,E2 -15178.69} C_VEL
LIN {X 0,Y 475.321,Z 313.477,A -85,B 0,C 180,E1 -15181.628,E2 -15181.628} C_VEL
LIN {X 0,Y 477.918,Z 325.947,A -85,B 0,C 180,E1 -15183.919,E2 -15183.919} C_VEL
LIN {X 0,Y 477.459,Z 332.79,A -85,B 0,C 180,E1 -15185.044,E2 -15185.044} C_VEL
LIN {X 0,Y 475.227,Z 355.557,A -85,B 0,C 180,E1 -15188.671,E2 -15188.671} C_VEL
LIN {X 0,Y 480.456,Z 385.381,A -85,B 0,C 180,E1 -15189.435,E2 -15189.435} C_VEL
LIN {X 0,Y 482.345,Z 400.297,A -85,B 0,C 180,E1 -15189.772,E2 -15189.772} C_VEL
LIN {X 0,Y 480.686,Z 493.47,A -85,B 0,C 180,E1 -15191.194,E2 -15191.194} C_VEL
LIN {X 0,Y 479.947,Z 508.235,A -85,B 0,C 180,E1 -15191.583,E2 -15191.583} C_VEL
LIN {X 0,Y 478.994,Z 520.635,A -85,B 0,C 180,E1 -15192.049,E2 -15192.049} C_VEL
LIN {X 0,Y 477.889,Z 534.16,A -85,B 0,C 180,E1 -15192.737,E2 -15192.737} C_VEL
LIN {X 0,Y 476.62,Z 546.929,A -85,B 0,C 180,E1 -15193.569,E2 -15193.569} C_VEL
LIN {X 0,Y 475.143,Z 559.73,A -85,B 0,C 180,E1 -15194.615,E2 -15194.615} C_VEL
LIN {X 0,Y 473.97,Z 570.219,A -85,B 0,C 180,E1 -15195.671,E2 -15195.671} C_VEL
LIN {X 0,Y 472.782,Z 580.675,A -85,B 0,C 180,E1 -15196.945,E2 -15196.945} C_VEL
LIN {X 0,Y 471.816,Z 590.398,A -85,B 0,C 180,E1 -15198.397,E2 -15198.397} C_VEL
LIN {X 0,Y 470.899,Z 598.721,A -85,B 0,C 180,E1 -15199.937,E2 -15199.937} C_VEL
LIN {X 0,Y 470.34,Z 605.261,A -85,B 0,C 180,E1 -15201.438,E2 -15201.438} C_VEL
LIN {X 0,Y 470.002,Z 611.107,A -85,B 0,C 180,E1 -15203.155,E2 -15203.155} C_VEL
LIN {X 0,Y 469.863,Z 618.194,A -85,B 0,C 180,E1 -15205.299,E2 -15205.299} C_VEL
LIN {X 0,Y 469.843,Z 621.42,A -85,B 0,C 180,E1 -15206.583,E2 -15206.583} C_VEL
LIN {X 0,Y 469.866,Z 624.367,A -85,B 0,C 180,E1 -15208.294,E2 -15208.294} C_VEL
LIN {X 0,Y 469.89,Z 625.831,A -85,B 0,C 180,E1 -15210.002,E2 -15210.002} C_VEL
LIN {X 0,Y 469.835,Z 625.832,A -85,B 0,C 180,E1 -15211.711,E2 -15211.711} C_VEL
LIN {X 0,Y 469.841,Z 624.357,A -85,B 0,C 180,E1 -15213.421,E2 -15213.421} C_VEL
LIN {X 0,Y 469.916,Z 621.422,A -85,B 0,C 180,E1 -15215.133,E2 -15215.133} C_VEL
LIN {X 0,Y 470.139,Z 616.962,A -85,B 0,C 180,E1 -15216.847,E2 -15216.847} C_VEL
LIN {X 0,Y 470.429,Z 612.536,A -85,B 0,C 180,E1 -15218.134,E2 -15218.134} C_VEL
LIN {X 0,Y 471.065,Z 606.069,A -85,B 0,C 180,E1 -15219.632,E2 -15219.632} C_VEL
LIN {X 0,Y 471.746,Z 598.03,A -85,B 0,C 180,E1 -15221.131,E2 -15221.131} C_VEL
LIN {X 0,Y 472.661,Z 589.622,A -85,B 0,C 180,E1 -15222.41,E2 -15222.41} C_VEL
LIN {X 0,Y 473.707,Z 579.527,A -85,B 0,C 180,E1 -15223.687,E2 -15223.687} C_VEL
LIN {X 0,Y 474.844,Z 568.352,A -85,B 0,C 180,E1 -15224.852,E2 -15224.852} C_VEL
LIN {X 0,Y 476.093,Z 555.892,A -85,B 0,C 180,E1 -15225.905,E2 -15225.905} C_VEL
LIN {X 0,Y 477.104,Z 545.381,A -85,B 0,C 180,E1 -15226.637,E2 -15226.637} C_VEL
LIN {X 0,Y 478.234,Z 531.428,A -85,B 0,C 180,E1 -15227.42,E2 -15227.42} C_VEL
LIN {X 0,Y 479.253,Z 517.041,A -85,B 0,C 180,E1 -15228.032,E2 -15228.032} C_VEL
LIN {X 0,Y 480.09,Z 502.653,A -85,B 0,C 180,E1 -15228.465,E2 -15228.465} C_VEL
LIN {X 0,Y 483.689,Z 400.437,A -85,B 0,C 180,E1 -15230.54,E2 -15230.54} C_VEL
LIN {X 0,Y 481.981,Z 382.027,A -85,B 0,C 180,E1 -15231.087,E2 -15231.087} C_VEL
LIN {X 0,Y 478.61,Z 359.027,A -85,B 0,C 180,E1 -15231.885,E2 -15231.885} C_VEL
LIN {X 0,Y 477.617,Z 352.997,A -85,B 0,C 180,E1 -15232.147,E2 -15232.147} C_VEL
LIN {X 0,Y 475.039,Z 330.34,A -85,B 0,C 180,E1 -15233.586,E2 -15233.586} C_VEL
LIN {X 0,Y 475.768,Z 319.53,A -85,B 0,C 180,E1 -15235.276,E2 -15235.276} C_VEL
LIN {X 0,Y 472.716,Z 303.053,A -85,B 0,C 180,E1 -15238.065,E2 -15238.065} C_VEL
LIN {X 0,Y 471.729,Z 298.283,A -85,B 0,C 180,E1 -15238.934,E2 -15238.934} C_VEL
LIN {X 0,Y 471.632,Z 298.289,A -85,B 0,C 180,E1 -15242.163,E2 -15242.163} C_VEL
LIN {X 0,Y 471.664,Z 298.292,A -85,B 0,C 180,E1 -15245.394,E2 -15245.394} C_VEL
LIN {X 0,Y 471.631,Z 298.294,A -85,B 0,C 180,E1 -15248.593,E2 -15248.593} C_VEL
LIN {X 0,Y 471.676,Z 298.288,A -85,B 0,C 180,E1 -15250.801,E2 -15250.801} C_VEL
LIN {X 0,Y 471.698,Z 298.284,A -85,B 0,C 180,E1 -15254.263,E2 -15254.263} C_VEL
LIN {X 0,Y 471.672,Z 298.288,A -85,B 0,C 180,E1 -15256.913,E2 -15256.913} C_VEL
LIN {X 0,Y 471.676,Z 298.29,A -85,B 0,C 180,E1 -15259.234,E2 -15259.234} C_VEL
LIN {X 0,Y 471.666,Z 298.293,A -85,B 0,C 180,E1 -15262.492,E2 -15262.492} C_VEL
LIN {X 0,Y 471.681,Z 298.287,A -85,B 0,C 180,E1 -15265.646,E2 -15265.646} C_VEL
LIN {X 0,Y 471.677,Z 298.289,A -85,B 0,C 180,E1 -15268.684,E2 -15268.684} C_VEL
LIN {X 0,Y 471.705,Z 298.284,A -85,B 0,C 180,E1 -15271.629,E2 -15271.629} C_VEL
LIN {X 0,Y 471.709,Z 298.289,A -85,B 0,C 180,E1 -15274.493,E2 -15274.493} C_VEL
LIN {X 0,Y 471.732,Z 298.287,A -85,B 0,C 180,E1 -15277.291,E2 -15277.291} C_VEL
LIN {X 0,Y 471.731,Z 298.293,A -85,B 0,C 180,E1 -15280.031,E2 -15280.031} C_VEL
LIN {X 0,Y 471.795,Z 298.424,A -85,B 0,C 180,E1 -15282.045,E2 -15282.045} C_VEL
LIN {X 0,Y 476.348,Z 313.233,A -85,B 0,C 180,E1 -15284.87,E2 -15284.87} C_VEL
LIN {X 0,Y 479.002,Z 324.767,A -85,B 0,C 180,E1 -15286.9,E2 -15286.9} C_VEL
LIN {X 0,Y 479.719,Z 330.106,A -85,B 0,C 180,E1 -15287.777,E2 -15287.777} C_VEL
LIN {X 0,Y 478.712,Z 345.477,A -85,B 0,C 180,E1 -15290.034,E2 -15290.034} C_VEL
LIN {X 0,Y 483.172,Z 365.803,A -85,B 0,C 180,E1 -15290.844,E2 -15290.844} C_VEL
LIN {X 0,Y 484.865,Z 375.502,A -85,B 0,C 180,E1 -15291.188,E2 -15291.188} C_VEL
LIN {X 0,Y 480.849,Z 486.401,A -85,B 0,C 180,E1 -15293.439,E2 -15293.439} C_VEL
LIN {X 0,Y 480.155,Z 499.994,A -85,B 0,C 180,E1 -15293.876,E2 -15293.876} C_VEL
LIN {X 0,Y 479.164,Z 514.012,A -85,B 0,C 180,E1 -15294.493,E2 -15294.493} C_VEL
LIN {X 0,Y 478.003,Z 527.847,A -85,B 0,C 180,E1 -15295.288,E2 -15295.288} C_VEL
LIN {X 0,Y 476.789,Z 540.56,A -85,B 0,C 180,E1 -15296.209,E2 -15296.209} C_VEL
LIN {X 0,Y 475.66,Z 552.242,A -85,B 0,C 180,E1 -15297.257,E2 -15297.257} C_VEL
LIN {X 0,Y 474.478,Z 563.72,A -85,B 0,C 180,E1 -15298.52,E2 -15298.52} C_VEL
LIN {X 0,Y 473.235,Z 573.277,A -85,B 0,C 180,E1 -15299.788,E2 -15299.788} C_VEL
LIN {X 0,Y 472.304,Z 581.21,A -85,B 0,C 180,E1 -15301.062,E2 -15301.062} C_VEL
LIN {X 0,Y 471.419,Z 588.83,A -85,B 0,C 180,E1 -15302.555,E2 -15302.555} C_VEL
LIN {X 0,Y 470.906,Z 594.104,A -85,B 0,C 180,E1 -15303.838,E2 -15303.838} C_VEL
LIN {X 0,Y 470.507,Z 599.265,A -85,B 0,C 180,E1 -15305.422,E2 -15305.422} C_VEL
LIN {X 0,Y 470.169,Z 602.727,A -85,B 0,C 180,E1 -15306.845,E2 -15306.845} C_VEL
LIN {X 0,Y 469.854,Z 605.554,A -85,B 0,C 180,E1 -15308.573,E2 -15308.573} C_VEL
LIN {X 0,Y 469.804,Z 606.917,A -85,B 0,C 180,E1 -15310.306,E2 -15310.306} C_VEL
LIN {X 0,Y 469.643,Z 606.79,A -85,B 0,C 180,E1 -15312.052,E2 -15312.052} C_VEL
LIN {X 0,Y 469.726,Z 605.165,A -85,B 0,C 180,E1 -15313.803,E2 -15313.803} C_VEL
LIN {X 0,Y 469.768,Z 602.002,A -85,B 0,C 180,E1 -15315.568,E2 -15315.568} C_VEL
LIN {X 0,Y 469.908,Z 598.534,A -85,B 0,C 180,E1 -15316.898,E2 -15316.898} C_VEL
LIN {X 0,Y 470.087,Z 594.05,A -85,B 0,C 180,E1 -15318.234,E2 -15318.234} C_VEL
LIN {X 0,Y 470.424,Z 587.363,A -85,B 0,C 180,E1 -15319.8,E2 -15319.8} C_VEL
LIN {X 0,Y 470.831,Z 578.894,A -85,B 0,C 180,E1 -15321.376,E2 -15321.376} C_VEL
LIN {X 0,Y 471.353,Z 569.917,A -85,B 0,C 180,E1 -15322.729,E2 -15322.729} C_VEL
LIN {X 0,Y 471.96,Z 559.896,A -85,B 0,C 180,E1 -15323.971,E2 -15323.971} C_VEL
LIN {X 0,Y 472.581,Z 550.117,A -85,B 0,C 180,E1 -15324.987,E2 -15324.987} C_VEL
LIN {X 0,Y 473.281,Z 538.324,A -85,B 0,C 180,E1 -15326.005,E2 -15326.005} C_VEL
LIN {X 0,Y 473.981,Z 525.446,A -85,B 0,C 180,E1 -15326.909,E2 -15326.909} C_VEL
LIN {X 0,Y 474.636,Z 511.395,A -85,B 0,C 180,E1 -15327.69,E2 -15327.69} C_VEL
LIN {X 0,Y 475.285,Z 497.078,A -85,B 0,C 180,E1 -15328.288,E2 -15328.288} C_VEL
LIN {X 0,Y 475.778,Z 482.848,A -85,B 0,C 180,E1 -15328.705,E2 -15328.705} C_VEL
LIN {X 0,Y 477.915,Z 371.198,A -85,B 0,C 180,E1 -15330.774,E2 -15330.774} C_VEL
LIN {X 0,Y 474.145,Z 343.622,A -85,B 0,C 180,E1 -15331.435,E2 -15331.435} C_VEL
LIN {X 0,Y 475.071,Z 322.865,A -85,B 0,C 180,E1 -15334.437,E2 -15334.437} C_VEL
LIN {X 0,Y 475.325,Z 316.895,A -85,B 0,C 180,E1 -15335.305,E2 -15335.305} C_VEL
LIN {X 0,Y 472.465,Z 301.976,A -85,B 0,C 180,E1 -15337.61,E2 -15337.61} C_VEL
LIN {X 0,Y 471.686,Z 298.29,A -85,B 0,C 180,E1 -15338.229,E2 -15338.229} C_VEL
LIN {X 0,Y 471.677,Z 298.288,A -85,B 0,C 180,E1 -15340.799,E2 -15340.799} C_VEL
LIN {X 0,Y 471.692,Z 298.29,A -85,B 0,C 180,E1 -15344.261,E2 -15344.261} C_VEL
LIN {X 0,Y 471.672,Z 298.287,A -85,B 0,C 180,E1 -15346.911,E2 -15346.911} C_VEL
LIN {X 0,Y 471.675,Z 298.285,A -85,B 0,C 180,E1 -15349.232,E2 -15349.232} C_VEL
LIN {X 0,Y 471.627,Z 298.296,A -85,B 0,C 180,E1 -15352.487,E2 -15352.487} C_VEL
LIN {X 0,Y 471.664,Z 298.288,A -85,B 0,C 180,E1 -15355.643,E2 -15355.643} C_VEL
LIN {X 0,Y 471.652,Z 298.29,A -85,B 0,C 180,E1 -15358.681,E2 -15358.681} C_VEL
LIN {X 0,Y 471.697,Z 298.285,A -85,B 0,C 180,E1 -15361.627,E2 -15361.627} C_VEL
LIN {X 0,Y 471.701,Z 298.282,A -85,B 0,C 180,E1 -15364.933,E2 -15364.933} C_VEL
LIN {X 0,Y 471.736,Z 298.283,A -85,B 0,C 180,E1 -15368.208,E2 -15368.208} C_VEL
LIN {X 0,Y 471.734,Z 298.278,A -85,B 0,C 180,E1 -15370.932,E2 -15370.932} C_VEL
LIN {X 0,Y 471.756,Z 298.279,A -85,B 0,C 180,E1 -15373.612,E2 -15373.612} C_VEL
LIN {X 0,Y 471.782,Z 298.275,A -85,B 0,C 180,E1 -15376.256,E2 -15376.256} C_VEL
LIN {X 0,Y 471.859,Z 298.262,A -85,B 0,C 180,E1 -15378.872,E2 -15378.872} C_VEL
LIN {X 0,Y 471.848,Z 298.29,A -85,B 0,C 180,E1 -15381.031,E2 -15381.031} C_VEL
LIN {X 0,Y 473.16,Z 305.269,A -85,B 0,C 180,E1 -15382.526,E2 -15382.526} C_VEL
LIN {X 0,Y 476.164,Z 315.623,A -85,B 0,C 180,E1 -15382.793,E2 -15382.793} C_VEL
LIN {X 0,Y 478.812,Z 329.109,A -85,B 0,C 180,E1 -15383.093,E2 -15383.093} C_VEL
LIN {X 0,Y 477.113,Z 441.215,A -85,B 0,C 180,E1 -15384.786,E2 -15384.786} C_VEL
LIN {X 0,Y 476.746,Z 455.531,A -85,B 0,C 180,E1 -15385.178,E2 -15385.178} C_VEL
LIN {X 0,Y 476.21,Z 469.308,A -85,B 0,C 180,E1 -15385.728,E2 -15385.728} C_VEL
LIN {X 0,Y 475.637,Z 482.128,A -85,B 0,C 180,E1 -15386.41,E2 -15386.41} C_VEL
LIN {X 0,Y 474.971,Z 494.583,A -85,B 0,C 180,E1 -15387.251,E2 -15387.251} C_VEL
LIN {X 0,Y 473.928,Z 506.979,A -85,B 0,C 180,E1 -15388.284,E2 -15388.284} C_VEL
LIN {X 0,Y 472.967,Z 511.637,A -85,B 0,C 180,E1 -15388.711,E2 -15388.711} C_VEL
LIN {X 0,Y 469.617,Z 518.93,A -85,B 0,C 180,E1 -15389.423,E2 -15389.423} C_VEL
LIN {X 0,Y 466.258,Z 525.747,A -85,B 0,C 180,E1 -15390.207,E2 -15390.207} C_VEL
LIN {X 0,Y 465.293,Z 529.657,A -85,B 0,C 180,E1 -15390.74,E2 -15390.74} C_VEL
LIN {X 0,Y 464.65,Z 538.531,A -85,B 0,C 180,E1 -15392.158,E2 -15392.158} C_VEL
LIN {X 0,Y 464.037,Z 545.274,A -85,B 0,C 180,E1 -15393.459,E2 -15393.459} C_VEL
LIN {X 0,Y 463.861,Z 550.667,A -85,B 0,C 180,E1 -15394.712,E2 -15394.712} C_VEL
LIN {X 0,Y 463.487,Z 555.433,A -85,B 0,C 180,E1 -15396.07,E2 -15396.07} C_VEL
LIN {X 0,Y 463.136,Z 560.166,A -85,B 0,C 180,E1 -15397.821,E2 -15397.821} C_VEL
LIN {X 0,Y 462.995,Z 563.388,A -85,B 0,C 180,E1 -15399.577,E2 -15399.577} C_VEL
LIN {X 0,Y 462.938,Z 565.227,A -85,B 0,C 180,E1 -15401.341,E2 -15401.341} C_VEL
LIN {X 0,Y 462.981,Z 565.72,A -85,B 0,C 180,E1 -15403.114,E2 -15403.114} C_VEL
LIN {X 0,Y 463.215,Z 564.853,A -85,B 0,C 180,E1 -15404.893,E2 -15404.893} C_VEL
LIN {X 0,Y 463.437,Z 562.604,A -85,B 0,C 180,E1 -15406.686,E2 -15406.686} C_VEL
LIN {X 0,Y 463.965,Z 558.885,A -85,B 0,C 180,E1 -15408.481,E2 -15408.481} C_VEL
LIN {X 0,Y 464.513,Z 555.018,A -85,B 0,C 180,E1 -15409.83,E2 -15409.83} C_VEL
LIN {X 0,Y 465.128,Z 550.185,A -85,B 0,C 180,E1 -15411.185,E2 -15411.185} C_VEL
LIN {X 0,Y 466.079,Z 543.114,A -85,B 0,C 180,E1 -15412.764,E2 -15412.764} C_VEL
LIN {X 0,Y 467.09,Z 535.646,A -85,B 0,C 180,E1 -15414.117,E2 -15414.117} C_VEL
LIN {X 0,Y 468.228,Z 526.576,A -85,B 0,C 180,E1 -15415.47,E2 -15415.47} C_VEL
LIN {X 0,Y 469.507,Z 516.5,A -85,B 0,C 180,E1 -15416.704,E2 -15416.704} C_VEL
LIN {X 0,Y 470.757,Z 505.369,A -85,B 0,C 180,E1 -15417.826,E2 -15417.826} C_VEL
LIN {X 0,Y 471.854,Z 494.159,A -85,B 0,C 180,E1 -15418.753,E2 -15418.753} C_VEL
LIN {X 0,Y 472.792,Z 482.977,A -85,B 0,C 180,E1 -15419.509,E2 -15419.509} C_VEL
LIN {X 0,Y 473.685,Z 469.332,A -85,B 0,C 180,E1 -15420.241,E2 -15420.241} C_VEL
LIN {X 0,Y 474.465,Z 455.181,A -85,B 0,C 180,E1 -15420.8,E2 -15420.8} C_VEL
LIN {X 0,Y 474.866,Z 441.988,A -85,B 0,C 180,E1 -15421.16,E2 -15421.16} C_VEL
LIN {X 0,Y 476.359,Z 362.546,A -85,B 0,C 180,E1 -15422.397,E2 -15422.397} C_VEL
LIN {X 0,Y 476.833,Z 332.508,A -85,B 0,C 180,E1 -15422.862,E2 -15422.862} C_VEL
LIN {X 0,Y 470.222,Z 315.768,A -85,B 0,C 180,E1 -15423.514,E2 -15423.514} C_VEL
LIN {X 0,Y 466.249,Z 306.718,A -85,B 0,C 180,E1 -15423.904,E2 -15423.904} C_VEL
LIN {X 0,Y 464.617,Z 299.171,A -85,B 0,C 180,E1 -15425.788,E2 -15425.788} C_VEL
LIN {X 0,Y 464.588,Z 299.168,A -85,B 0,C 180,E1 -15429.285,E2 -15429.285} C_VEL
LIN {X 0,Y 464.617,Z 299.17,A -85,B 0,C 180,E1 -15432.716,E2 -15432.716} C_VEL
LIN {X 0,Y 464.651,Z 299.149,A -85,B 0,C 180,E1 -15435.11,E2 -15435.11} C_VEL
LIN {X 0,Y 464.609,Z 299.17,A -85,B 0,C 180,E1 -15438.445,E2 -15438.445} C_VEL
LIN {X 0,Y 464.599,Z 299.172,A -85,B 0,C 180,E1 -15441.621,E2 -15441.621} C_VEL
LIN {X 0,Y 464.619,Z 299.144,A -85,B 0,C 180,E1 -15444.492,E2 -15444.492} C_VEL
LIN {X 0,Y 464.622,Z 299.17,A -85,B 0,C 180,E1 -15447.584,E2 -15447.584} C_VEL
LIN {X 0,Y 464.627,Z 299.167,A -85,B 0,C 180,E1 -15450.166,E2 -15450.166} C_VEL
LIN {X 0,Y 464.677,Z 299.151,A -85,B 0,C 180,E1 -15453.114,E2 -15453.114} C_VEL
LIN {X 0,Y 464.601,Z 299.162,A -85,B 0,C 180,E1 -15455.98,E2 -15455.98} C_VEL
LIN {X 0,Y 464.679,Z 299.161,A -85,B 0,C 180,E1 -15459.151,E2 -15459.151} C_VEL
LIN {X 0,Y 464.664,Z 299.157,A -85,B 0,C 180,E1 -15462.453,E2 -15462.453} C_VEL
LIN {X 0,Y 464.745,Z 299.146,A -85,B 0,C 180,E1 -15465.154,E2 -15465.154} C_VEL
LIN {X 0,Y 464.781,Z 299.145,A -85,B 0,C 180,E1 -15468.386,E2 -15468.386} C_VEL
LIN {X 0,Y 464.837,Z 299.134,A -85,B 0,C 180,E1 -15472.206,E2 -15472.206} C_VEL
LIN {X 0,Y 464.887,Z 299.134,A -85,B 0,C 180,E1 -15474.813,E2 -15474.813} C_VEL
LIN {X 0,Y 464.747,Z 299.145,A -85,B 0,C 180,E1 -15477.409,E2 -15477.409} C_VEL
LIN {X 0,Y 464.941,Z 299.123,A -85,B 0,C 180,E1 -15480,E2 -15480} C_VEL
LIN {X 0,Y 464.916,Z 299.127,A -85,B 0,C 180,E1 -15484.32,E2 -15484.32} C_VEL
LIN {X 0,Y 464.83,Z 299.13,A -85,B 0,C 180,E1 -15486.924,E2 -15486.924} C_VEL
LIN {X 0,Y 464.798,Z 299.142,A -85,B 0,C 180,E1 -15490.419,E2 -15490.419} C_VEL
LIN {X 0,Y 464.745,Z 299.141,A -85,B 0,C 180,E1 -15493.066,E2 -15493.066} C_VEL
LIN {X 0,Y 464.735,Z 299.147,A -85,B 0,C 180,E1 -15495.741,E2 -15495.741} C_VEL
LIN {X 0,Y 464.697,Z 299.147,A -85,B 0,C 180,E1 -15498.454,E2 -15498.454} C_VEL
LIN {X 0,Y 464.653,Z 299.154,A -85,B 0,C 180,E1 -15501.21,E2 -15501.21} C_VEL
LIN {X 0,Y 464.601,Z 299.167,A -85,B 0,C 180,E1 -15504.02,E2 -15504.02} C_VEL
LIN {X 0,Y 464.651,Z 299.16,A -85,B 0,C 180,E1 -15507.208,E2 -15507.208} C_VEL
LIN {X 0,Y 464.639,Z 299.161,A -85,B 0,C 180,E1 -15509.833,E2 -15509.833} C_VEL
LIN {X 0,Y 464.639,Z 299.163,A -85,B 0,C 180,E1 -15512.868,E2 -15512.868} C_VEL
LIN {X 0,Y 464.681,Z 299.131,A -85,B 0,C 180,E1 -15516.006,E2 -15516.006} C_VEL
LIN {X 0,Y 464.666,Z 299.159,A -85,B 0,C 180,E1 -15519.28,E2 -15519.28} C_VEL
LIN {X 0,Y 464.622,Z 299.164,A -85,B 0,C 180,E1 -15522.719,E2 -15522.719} C_VEL
LIN {X 0,Y 464.666,Z 299.156,A -85,B 0,C 180,E1 -15525.112,E2 -15525.112} C_VEL
LIN {X 0,Y 464.645,Z 299.166,A -85,B 0,C 180,E1 -15528.452,E2 -15528.452} C_VEL
LIN {X 0,Y 464.665,Z 299.161,A -85,B 0,C 180,E1 -15530.723,E2 -15530.723} C_VEL
LIN {X 0,Y 464.687,Z 299.155,A -85,B 0,C 180,E1 -15533.998,E2 -15533.998} C_VEL
LIN {X 0,Y 464.643,Z 299.169,A -85,B 0,C 180,E1 -15537.136,E2 -15537.136} C_VEL
LIN {X 0,Y 464.706,Z 299.275,A -85,B 0,C 180,E1 -15538.321,E2 -15538.321} C_VEL
LIN {X 0,Y 468.405,Z 314.861,A -85,B 0,C 180,E1 -15541.414,E2 -15541.414} C_VEL
LIN {X 0,Y 471,Z 327.263,A -85,B 0,C 180,E1 -15543.744,E2 -15543.744} C_VEL
LIN {X 0,Y 470.878,Z 331.418,A -85,B 0,C 180,E1 -15544.447,E2 -15544.447} C_VEL
LIN {X 0,Y 468.89,Z 349.537,A -85,B 0,C 180,E1 -15547.403,E2 -15547.403} C_VEL
LIN {X 0,Y 468.43,Z 354.946,A -85,B 0,C 180,E1 -15548.28,E2 -15548.28} C_VEL
LIN {X 0,Y 473.734,Z 385.06,A -85,B 0,C 180,E1 -15549.073,E2 -15549.073} C_VEL
LIN {X 0,Y 475.833,Z 400.428,A -85,B 0,C 180,E1 -15549.436,E2 -15549.436} C_VEL
LIN {X 0,Y 474.129,Z 492.961,A -85,B 0,C 180,E1 -15550.868,E2 -15550.868} C_VEL
LIN {X 0,Y 473.389,Z 507.382,A -85,B 0,C 180,E1 -15551.249,E2 -15551.249} C_VEL
LIN {X 0,Y 472.289,Z 521.294,A -85,B 0,C 180,E1 -15551.785,E2 -15551.785} C_VEL
LIN {X 0,Y 471.138,Z 534.587,A -85,B 0,C 180,E1 -15552.481,E2 -15552.481} C_VEL
LIN {X 0,Y 469.834,Z 547.193,A -85,B 0,C 180,E1 -15553.325,E2 -15553.325} C_VEL
LIN {X 0,Y 468.497,Z 558.704,A -85,B 0,C 180,E1 -15554.28,E2 -15554.28} C_VEL
LIN {X 0,Y 467.303,Z 568.322,A -85,B 0,C 180,E1 -15555.24,E2 -15555.24} C_VEL
LIN {X 0,Y 466.019,Z 579.021,A -85,B 0,C 180,E1 -15556.53,E2 -15556.53} C_VEL
LIN {X 0,Y 465.078,Z 587.889,A -85,B 0,C 180,E1 -15557.83,E2 -15557.83} C_VEL
LIN {X 0,Y 464.153,Z 596.423,A -85,B 0,C 180,E1 -15559.349,E2 -15559.349} C_VEL
LIN {X 0,Y 463.458,Z 603.333,A -85,B 0,C 180,E1 -15560.871,E2 -15560.871} C_VEL
LIN {X 0,Y 462.976,Z 609.568,A -85,B 0,C 180,E1 -15562.614,E2 -15562.614} C_VEL
LIN {X 0,Y 462.877,Z 613.518,A -85,B 0,C 180,E1 -15563.922,E2 -15563.922} C_VEL
LIN {X 0,Y 462.795,Z 617.763,A -85,B 0,C 180,E1 -15565.227,E2 -15565.227} C_VEL
LIN {X 0,Y 462.751,Z 621.07,A -85,B 0,C 180,E1 -15566.531,E2 -15566.531} C_VEL
LIN {X 0,Y 462.778,Z 624.094,A -85,B 0,C 180,E1 -15568.267,E2 -15568.267} C_VEL
LIN {X 0,Y 462.796,Z 625.626,A -85,B 0,C 180,E1 -15570.002,E2 -15570.002} C_VEL
LIN {X 0,Y 462.749,Z 625.702,A -85,B 0,C 180,E1 -15571.737,E2 -15571.737} C_VEL
LIN {X 0,Y 462.75,Z 624.321,A -85,B 0,C 180,E1 -15573.473,E2 -15573.473} C_VEL
LIN {X 0,Y 462.845,Z 621.452,A -85,B 0,C 180,E1 -15575.212,E2 -15575.212} C_VEL
LIN {X 0,Y 463.067,Z 617.063,A -85,B 0,C 180,E1 -15576.952,E2 -15576.952} C_VEL
LIN {X 0,Y 463.371,Z 612.72,A -85,B 0,C 180,E1 -15578.258,E2 -15578.258} C_VEL
LIN {X 0,Y 464.063,Z 606.334,A -85,B 0,C 180,E1 -15579.778,E2 -15579.778} C_VEL
LIN {X 0,Y 464.786,Z 598.38,A -85,B 0,C 180,E1 -15581.3,E2 -15581.3} C_VEL
LIN {X 0,Y 465.733,Z 590.096,A -85,B 0,C 180,E1 -15582.598,E2 -15582.598} C_VEL
LIN {X 0,Y 466.861,Z 580.127,A -85,B 0,C 180,E1 -15583.892,E2 -15583.892} C_VEL
LIN {X 0,Y 468.048,Z 569.108,A -85,B 0,C 180,E1 -15585.073,E2 -15585.073} C_VEL
LIN {X 0,Y 469.341,Z 556.956,A -85,B 0,C 180,E1 -15586.14,E2 -15586.14} C_VEL
LIN {X 0,Y 470.539,Z 545.054,A -85,B 0,C 180,E1 -15586.988,E2 -15586.988} C_VEL
LIN {X 0,Y 471.647,Z 532.145,A -85,B 0,C 180,E1 -15587.727,E2 -15587.727} C_VEL
LIN {X 0,Y 472.741,Z 518.063,A -85,B 0,C 180,E1 -15588.344,E2 -15588.344} C_VEL
LIN {X 0,Y 473.616,Z 503.634,A -85,B 0,C 180,E1 -15588.802,E2 -15588.802} C_VEL
LIN {X 0,Y 477.458,Z 400.818,A -85,B 0,C 180,E1 -15590.948,E2 -15590.948} C_VEL
LIN {X 0,Y 475.9,Z 383.781,A -85,B 0,C 180,E1 -15591.47,E2 -15591.47} C_VEL
LIN {X 0,Y 472.683,Z 361.202,A -85,B 0,C 180,E1 -15592.276,E2 -15592.276} C_VEL
LIN {X 0,Y 471.429,Z 354.176,A -85,B 0,C 180,E1 -15592.56,E2 -15592.56} C_VEL
LIN {X 0,Y 469.053,Z 332.539,A -85,B 0,C 180,E1 -15593.982,E2 -15593.982} C_VEL
LIN {X 0,Y 468.401,Z 326.553,A -85,B 0,C 180,E1 -15594.432,E2 -15594.432} C_VEL
LIN {X 0,Y 468.775,Z 320.206,A -85,B 0,C 180,E1 -15595.443,E2 -15595.443} C_VEL
LIN {X 0,Y 465.616,Z 303.726,A -85,B 0,C 180,E1 -15598.287,E2 -15598.287} C_VEL
LIN {X 0,Y 464.683,Z 299.162,A -85,B 0,C 180,E1 -15599.117,E2 -15599.117} C_VEL
LIN {X 0,Y 464.601,Z 299.164,A -85,B 0,C 180,E1 -15602.406,E2 -15602.406} C_VEL
LIN {X 0,Y 464.608,Z 299.17,A -85,B 0,C 180,E1 -15605.501,E2 -15605.501} C_VEL
LIN {X 0,Y 464.588,Z 299.172,A -85,B 0,C 180,E1 -15608.373,E2 -15608.373} C_VEL
LIN {X 0,Y 464.626,Z 299.169,A -85,B 0,C 180,E1 -15611.555,E2 -15611.555} C_VEL
LIN {X 0,Y 464.664,Z 299.162,A -85,B 0,C 180,E1 -15614.888,E2 -15614.888} C_VEL
LIN {X 0,Y 464.607,Z 299.169,A -85,B 0,C 180,E1 -15617.625,E2 -15617.625} C_VEL
LIN {X 0,Y 464.61,Z 299.171,A -85,B 0,C 180,E1 -15620.714,E2 -15620.714} C_VEL
LIN {X 0,Y 464.653,Z 299.164,A -85,B 0,C 180,E1 -15623.991,E2 -15623.991} C_VEL
LIN {X 0,Y 464.623,Z 299.166,A -85,B 0,C 180,E1 -15627.131,E2 -15627.131} C_VEL
LIN {X 0,Y 464.649,Z 299.164,A -85,B 0,C 180,E1 -15630.168,E2 -15630.168} C_VEL
LIN {X 0,Y 464.675,Z 299.163,A -85,B 0,C 180,E1 -15633.114,E2 -15633.114} C_VEL
LIN {X 0,Y 464.631,Z 299.172,A -85,B 0,C 180,E1 -15635.981,E2 -15635.981} C_VEL
LIN {X 0,Y 464.711,Z 299.166,A -85,B 0,C 180,E1 -15639.152,E2 -15639.152} C_VEL
LIN {X 0,Y 464.715,Z 299.318,A -85,B 0,C 180,E1 -15641.405,E2 -15641.405} C_VEL
LIN {X 0,Y 468.616,Z 311.489,A -85,B 0,C 180,E1 -15643.84,E2 -15643.84} C_VEL
LIN {X 0,Y 471.136,Z 320.752,A -85,B 0,C 180,E1 -15645.558,E2 -15645.558} C_VEL
LIN {X 0,Y 473.211,Z 331.512,A -85,B 0,C 180,E1 -15647.438,E2 -15647.438} C_VEL
LIN {X 0,Y 472.327,Z 345.708,A -85,B 0,C 180,E1 -15649.547,E2 -15649.547} C_VEL
LIN {X 0,Y 476.678,Z 365.353,A -85,B 0,C 180,E1 -15650.371,E2 -15650.371} C_VEL
LIN {X 0,Y 478.658,Z 376.97,A -85,B 0,C 180,E1 -15650.797,E2 -15650.797} C_VEL
LIN {X 0,Y 474.475,Z 486.039,A -85,B 0,C 180,E1 -15653.058,E2 -15653.058} C_VEL
LIN {X 0,Y 473.75,Z 499.098,A -85,B 0,C 180,E1 -15653.474,E2 -15653.474} C_VEL
LIN {X 0,Y 472.73,Z 513.812,A -85,B 0,C 180,E1 -15654.126,E2 -15654.126} C_VEL
LIN {X 0,Y 471.531,Z 527.039,A -85,B 0,C 180,E1 -15654.887,E2 -15654.887} C_VEL
LIN {X 0,Y 470.283,Z 540.116,A -85,B 0,C 180,E1 -15655.836,E2 -15655.836} C_VEL
LIN {X 0,Y 469.041,Z 551.932,A -85,B 0,C 180,E1 -15656.897,E2 -15656.897} C_VEL
LIN {X 0,Y 467.868,Z 562.611,A -85,B 0,C 180,E1 -15658.07,E2 -15658.07} C_VEL
LIN {X 0,Y 466.596,Z 572.362,A -85,B 0,C 180,E1 -15659.355,E2 -15659.355} C_VEL
LIN {X 0,Y 465.535,Z 580.484,A -85,B 0,C 180,E1 -15660.647,E2 -15660.647} C_VEL
LIN {X 0,Y 464.612,Z 588.244,A -85,B 0,C 180,E1 -15662.16,E2 -15662.16} C_VEL
LIN {X 0,Y 463.944,Z 593.681,A -85,B 0,C 180,E1 -15663.462,E2 -15663.462} C_VEL
LIN {X 0,Y 463.641,Z 598.103,A -85,B 0,C 180,E1 -15664.766,E2 -15664.766} C_VEL
LIN {X 0,Y 463.273,Z 601.595,A -85,B 0,C 180,E1 -15666.075,E2 -15666.075} C_VEL
LIN {X 0,Y 462.848,Z 604.938,A -85,B 0,C 180,E1 -15667.828,E2 -15667.828} C_VEL
LIN {X 0,Y 462.738,Z 606.76,A -85,B 0,C 180,E1 -15669.585,E2 -15669.585} C_VEL
LIN {X 0,Y 462.68,Z 607.131,A -85,B 0,C 180,E1 -15670.467,E2 -15670.467} C_VEL
LIN {X 0,Y 462.536,Z 606.775,A -85,B 0,C 180,E1 -15672.24,E2 -15672.24} C_VEL
LIN {X 0,Y 462.651,Z 604.932,A -85,B 0,C 180,E1 -15674.019,E2 -15674.019} C_VEL
LIN {X 0,Y 462.653,Z 603.435,A -85,B 0,C 180,E1 -15674.914,E2 -15674.914} C_VEL
LIN {X 0,Y 462.739,Z 600.384,A -85,B 0,C 180,E1 -15676.262,E2 -15676.262} C_VEL
LIN {X 0,Y 462.913,Z 596.368,A -85,B 0,C 180,E1 -15677.615,E2 -15677.615} C_VEL
LIN {X 0,Y 463.12,Z 591.271,A -85,B 0,C 180,E1 -15678.976,E2 -15678.976} C_VEL
LIN {X 0,Y 463.492,Z 584.402,A -85,B 0,C 180,E1 -15680.449,E2 -15680.449} C_VEL
LIN {X 0,Y 463.952,Z 575.796,A -85,B 0,C 180,E1 -15681.941,E2 -15681.941} C_VEL
LIN {X 0,Y 464.541,Z 566.101,A -85,B 0,C 180,E1 -15683.316,E2 -15683.316} C_VEL
LIN {X 0,Y 465.17,Z 555.224,A -85,B 0,C 180,E1 -15684.581,E2 -15684.581} C_VEL
LIN {X 0,Y 465.912,Z 544.022,A -85,B 0,C 180,E1 -15685.651,E2 -15685.651} C_VEL
LIN {X 0,Y 466.619,Z 531.355,A -85,B 0,C 180,E1 -15686.645,E2 -15686.645} C_VEL
LIN {X 0,Y 467.322,Z 517.652,A -85,B 0,C 180,E1 -15687.505,E2 -15687.505} C_VEL
LIN {X 0,Y 468.011,Z 503.755,A -85,B 0,C 180,E1 -15688.177,E2 -15688.177} C_VEL
LIN {X 0,Y 468.63,Z 488.953,A -85,B 0,C 180,E1 -15688.696,E2 -15688.696} C_VEL
LIN {X 0,Y 469.023,Z 472.834,A -85,B 0,C 180,E1 -15689.067,E2 -15689.067} C_VEL
LIN {X 0,Y 470.976,Z 371.902,A -85,B 0,C 180,E1 -15690.959,E2 -15690.959} C_VEL
LIN {X 0,Y 467.212,Z 343.651,A -85,B 0,C 180,E1 -15691.649,E2 -15691.649} C_VEL
LIN {X 0,Y 468.242,Z 321.419,A -85,B 0,C 180,E1 -15694.903,E2 -15694.903} C_VEL
LIN {X 0,Y 468.317,Z 317.887,A -85,B 0,C 180,E1 -15695.42,E2 -15695.42} C_VEL
LIN {X 0,Y 465.453,Z 303.026,A -85,B 0,C 180,E1 -15697.741,E2 -15697.741} C_VEL
LIN {X 0,Y 464.64,Z 299.168,A -85,B 0,C 180,E1 -15698.379,E2 -15698.379} C_VEL
LIN {X 0,Y 464.633,Z 299.162,A -85,B 0,C 180,E1 -15701.553,E2 -15701.553} C_VEL
LIN {X 0,Y 464.662,Z 299.16,A -85,B 0,C 180,E1 -15704.886,E2 -15704.886} C_VEL
LIN {X 0,Y 464.606,Z 299.166,A -85,B 0,C 180,E1 -15707.623,E2 -15707.623} C_VEL
LIN {X 0,Y 464.604,Z 299.168,A -85,B 0,C 180,E1 -15710.712,E2 -15710.712} C_VEL
LIN {X 0,Y 464.581,Z 299.174,A -85,B 0,C 180,E1 -15713.983,E2 -15713.983} C_VEL
LIN {X 0,Y 464.627,Z 299.17,A -85,B 0,C 180,E1 -15716.095,E2 -15716.095} C_VEL
LIN {X 0,Y 464.613,Z 299.165,A -85,B 0,C 180,E1 -15719.241,E2 -15719.241} C_VEL
LIN {X 0,Y 464.645,Z 299.167,A -85,B 0,C 180,E1 -15722.138,E2 -15722.138} C_VEL
LIN {X 0,Y 464.658,Z 299.159,A -85,B 0,C 180,E1 -15725.032,E2 -15725.032} C_VEL
LIN {X 0,Y 464.683,Z 299.162,A -85,B 0,C 180,E1 -15727.86,E2 -15727.86} C_VEL
LIN {X 0,Y 464.686,Z 299.156,A -85,B 0,C 180,E1 -15730.631,E2 -15730.631} C_VEL
LIN {X 0,Y 464.703,Z 299.155,A -85,B 0,C 180,E1 -15733.356,E2 -15733.356} C_VEL
LIN {X 0,Y 464.73,Z 299.156,A -85,B 0,C 180,E1 -15736.043,E2 -15736.043} C_VEL
LIN {X 0,Y 464.804,Z 299.141,A -85,B 0,C 180,E1 -15738.7,E2 -15738.7} C_VEL
LIN {X 0,Y 464.847,Z 299.331,A -85,B 0,C 180,E1 -15740.895,E2 -15740.895} C_VEL
LIN {X 0,Y 466.015,Z 305.613,A -85,B 0,C 180,E1 -15742.271,E2 -15742.271} C_VEL
LIN {X 0,Y 469.507,Z 317.376,A -85,B 0,C 180,E1 -15742.585,E2 -15742.585} C_VEL
LIN {X 0,Y 471.992,Z 330.344,A -85,B 0,C 180,E1 -15742.876,E2 -15742.876} C_VEL
LIN {X 0,Y 470.239,Z 441.468,A -85,B 0,C 180,E1 -15744.576,E2 -15744.576} C_VEL
LIN {X 0,Y 469.862,Z 455.834,A -85,B 0,C 180,E1 -15744.974,E2 -15744.974} C_VEL
LIN {X 0,Y 469.347,Z 469.075,A -85,B 0,C 180,E1 -15745.504,E2 -15745.504} C_VEL
LIN {X 0,Y 468.699,Z 482.909,A -85,B 0,C 180,E1 -15746.249,E2 -15746.249} C_VEL
LIN {X 0,Y 467.984,Z 495.302,A -85,B 0,C 180,E1 -15747.102,E2 -15747.102} C_VEL
LIN {X 0,Y 466.952,Z 507.445,A -85,B 0,C 180,E1 -15748.133,E2 -15748.133} C_VEL
LIN {X 0,Y 466.42,Z 517.073,A -85,B 0,C 180,E1 -15749.137,E2 -15749.137} C_VEL
LIN {X 0,Y 465.478,Z 527.471,A -85,B 0,C 180,E1 -15750.429,E2 -15750.429} C_VEL
LIN {X 0,Y 465.293,Z 529.657,A -85,B 0,C 180,E1 -15750.74,E2 -15750.74} C_VEL
LIN {X 0,Y 464.322,Z 533.453,A -85,B 0,C 180,E1 -15751.292,E2 -15751.292} C_VEL
LIN {X 0,Y 460.958,Z 539.265,A -85,B 0,C 180,E1 -15752.199,E2 -15752.199} C_VEL
LIN {X 0,Y 457.716,Z 544.615,A -85,B 0,C 180,E1 -15753.161,E2 -15753.161} C_VEL
LIN {X 0,Y 456.94,Z 547.525,A -85,B 0,C 180,E1 -15753.791,E2 -15753.791} C_VEL
LIN {X 0,Y 456.628,Z 553.369,A -85,B 0,C 180,E1 -15755.279,E2 -15755.279} C_VEL
LIN {X 0,Y 456.23,Z 558.762,A -85,B 0,C 180,E1 -15757.053,E2 -15757.053} C_VEL
LIN {X 0,Y 455.938,Z 562.595,A -85,B 0,C 180,E1 -15758.835,E2 -15758.835} C_VEL
LIN {X 0,Y 455.896,Z 565.013,A -85,B 0,C 180,E1 -15760.622,E2 -15760.622} C_VEL
LIN {X 0,Y 455.872,Z 566.085,A -85,B 0,C 180,E1 -15762.42,E2 -15762.42} C_VEL
LIN {X 0,Y 456.062,Z 565.801,A -85,B 0,C 180,E1 -15764.223,E2 -15764.223} C_VEL
LIN {X 0,Y 456.256,Z 564.154,A -85,B 0,C 180,E1 -15766.039,E2 -15766.039} C_VEL
LIN {X 0,Y 456.745,Z 561.078,A -85,B 0,C 180,E1 -15767.859,E2 -15767.859} C_VEL
LIN {X 0,Y 457.182,Z 557.729,A -85,B 0,C 180,E1 -15769.23,E2 -15769.23} C_VEL
LIN {X 0,Y 457.82,Z 553.468,A -85,B 0,C 180,E1 -15770.6,E2 -15770.6} C_VEL
LIN {X 0,Y 458.636,Z 547.158,A -85,B 0,C 180,E1 -15772.207,E2 -15772.207} C_VEL
LIN {X 0,Y 459.687,Z 540.048,A -85,B 0,C 180,E1 -15773.654,E2 -15773.654} C_VEL
LIN {X 0,Y 460.92,Z 530.825,A -85,B 0,C 180,E1 -15775.18,E2 -15775.18} C_VEL
LIN {X 0,Y 462.239,Z 520.859,A -85,B 0,C 180,E1 -15776.52,E2 -15776.52} C_VEL
LIN {X 0,Y 463.539,Z 510.304,A -85,B 0,C 180,E1 -15777.685,E2 -15777.685} C_VEL
LIN {X 0,Y 464.767,Z 499.038,A -85,B 0,C 180,E1 -15778.708,E2 -15778.708} C_VEL
LIN {X 0,Y 465.943,Z 486.387,A -85,B 0,C 180,E1 -15779.636,E2 -15779.636} C_VEL
LIN {X 0,Y 467,Z 472.863,A -85,B 0,C 180,E1 -15780.409,E2 -15780.409} C_VEL
LIN {X 0,Y 467.689,Z 460.406,A -85,B 0,C 180,E1 -15780.957,E2 -15780.957} C_VEL
LIN {X 0,Y 468.233,Z 447.018,A -85,B 0,C 180,E1 -15781.381,E2 -15781.381} C_VEL
LIN {X 0,Y 468.535,Z 430.552,A -85,B 0,C 180,E1 -15781.704,E2 -15781.704} C_VEL
LIN {X 0,Y 470.472,Z 334.203,A -85,B 0,C 180,E1 -15783.193,E2 -15783.193} C_VEL
LIN {X 0,Y 463.704,Z 317.603,A -85,B 0,C 180,E1 -15783.868,E2 -15783.868} C_VEL
LIN {X 0,Y 459.117,Z 307.089,A -85,B 0,C 180,E1 -15784.341,E2 -15784.341} C_VEL
LIN {X 0,Y 457.55,Z 300.05,A -85,B 0,C 180,E1 -15786.115,E2 -15786.115} C_VEL
LIN {X 0,Y 457.546,Z 300.043,A -85,B 0,C 180,E1 -15788.874,E2 -15788.874} C_VEL
LIN {X 0,Y 457.586,Z 300.041,A -85,B 0,C 180,E1 -15792.336,E2 -15792.336} C_VEL
LIN {X 0,Y 457.594,Z 300.028,A -85,B 0,C 180,E1 -15795.241,E2 -15795.241} C_VEL
LIN {X 0,Y 457.57,Z 300.046,A -85,B 0,C 180,E1 -15798.594,E2 -15798.594} C_VEL
LIN {X 0,Y 457.561,Z 300.046,A -85,B 0,C 180,E1 -15801.322,E2 -15801.322} C_VEL
LIN {X 0,Y 457.585,Z 300.019,A -85,B 0,C 180,E1 -15804.431,E2 -15804.431} C_VEL
LIN {X 0,Y 457.59,Z 300.046,A -85,B 0,C 180,E1 -15807.605,E2 -15807.605} C_VEL
LIN {X 0,Y 457.611,Z 300.039,A -85,B 0,C 180,E1 -15810.741,E2 -15810.741} C_VEL
LIN {X 0,Y 457.621,Z 300.036,A -85,B 0,C 180,E1 -15813.648,E2 -15813.648} C_VEL
LIN {X 0,Y 457.595,Z 300.031,A -85,B 0,C 180,E1 -15816.689,E2 -15816.689} C_VEL
LIN {X 0,Y 457.638,Z 300.04,A -85,B 0,C 180,E1 -15819.389,E2 -15819.389} C_VEL
LIN {X 0,Y 457.618,Z 300.036,A -85,B 0,C 180,E1 -15822.174,E2 -15822.174} C_VEL
LIN {X 0,Y 457.699,Z 300.027,A -85,B 0,C 180,E1 -15824.92,E2 -15824.92} C_VEL
LIN {X 0,Y 457.729,Z 300.024,A -85,B 0,C 180,E1 -15828.525,E2 -15828.525} C_VEL
LIN {X 0,Y 457.788,Z 300.012,A -85,B 0,C 180,E1 -15832.085,E2 -15832.085} C_VEL
LIN {X 0,Y 457.839,Z 300.011,A -85,B 0,C 180,E1 -15834.733,E2 -15834.733} C_VEL
LIN {X 0,Y 457.724,Z 300.019,A -85,B 0,C 180,E1 -15837.369,E2 -15837.369} C_VEL
LIN {X 0,Y 457.895,Z 300.001,A -85,B 0,C 180,E1 -15840,E2 -15840} C_VEL
LIN {X 0,Y 457.885,Z 300.004,A -85,B 0,C 180,E1 -15844.387,E2 -15844.387} C_VEL
LIN {X 0,Y 457.799,Z 300.004,A -85,B 0,C 180,E1 -15847.031,E2 -15847.031} C_VEL
LIN {X 0,Y 457.78,Z 300.018,A -85,B 0,C 180,E1 -15850.58,E2 -15850.58} C_VEL
LIN {X 0,Y 457.695,Z 300.02,A -85,B 0,C 180,E1 -15853.271,E2 -15853.271} C_VEL
LIN {X 0,Y 457.664,Z 300.028,A -85,B 0,C 180,E1 -15855.991,E2 -15855.991} C_VEL
LIN {X 0,Y 457.632,Z 300.031,A -85,B 0,C 180,E1 -15858.749,E2 -15858.749} C_VEL
LIN {X 0,Y 457.615,Z 300.029,A -85,B 0,C 180,E1 -15861.553,E2 -15861.553} C_VEL
LIN {X 0,Y 457.563,Z 300.047,A -85,B 0,C 180,E1 -15864.414,E2 -15864.414} C_VEL
LIN {X 0,Y 457.602,Z 300.037,A -85,B 0,C 180,E1 -15867.409,E2 -15867.409} C_VEL
LIN {X 0,Y 457.617,Z 300.034,A -85,B 0,C 180,E1 -15870.339,E2 -15870.339} C_VEL
LIN {X 0,Y 457.603,Z 300.036,A -85,B 0,C 180,E1 -15873.439,E2 -15873.439} C_VEL
LIN {X 0,Y 457.64,Z 300.014,A -85,B 0,C 180,E1 -15876.649,E2 -15876.649} C_VEL
LIN {X 0,Y 457.632,Z 300.036,A -85,B 0,C 180,E1 -15880.004,E2 -15880.004} C_VEL
LIN {X 0,Y 457.585,Z 300.041,A -85,B 0,C 180,E1 -15883.538,E2 -15883.538} C_VEL
LIN {X 0,Y 457.586,Z 300.045,A -85,B 0,C 180,E1 -15886.466,E2 -15886.466} C_VEL
LIN {X 0,Y 457.586,Z 300.042,A -85,B 0,C 180,E1 -15888.84,E2 -15888.84} C_VEL
LIN {X 0,Y 457.601,Z 300.04,A -85,B 0,C 180,E1 -15891.32,E2 -15891.32} C_VEL
LIN {X 0,Y 457.629,Z 300.039,A -85,B 0,C 180,E1 -15894.438,E2 -15894.438} C_VEL
LIN {X 0,Y 457.658,Z 300.177,A -85,B 0,C 180,E1 -15897.937,E2 -15897.937} C_VEL
LIN {X 0,Y 461.422,Z 315.946,A -85,B 0,C 180,E1 -15901.135,E2 -15901.135} C_VEL
LIN {X 0,Y 464.097,Z 328.591,A -85,B 0,C 180,E1 -15903.565,E2 -15903.565} C_VEL
LIN {X 0,Y 464.04,Z 332.74,A -85,B 0,C 180,E1 -15904.283,E2 -15904.283} C_VEL
LIN {X 0,Y 462.009,Z 350.709,A -85,B 0,C 180,E1 -15907.26,E2 -15907.26} C_VEL
LIN {X 0,Y 461.689,Z 354.369,A -85,B 0,C 180,E1 -15907.865,E2 -15907.865} C_VEL
LIN {X 0,Y 466.69,Z 382.157,A -85,B 0,C 180,E1 -15908.636,E2 -15908.636} C_VEL
LIN {X 0,Y 469.283,Z 400.63,A -85,B 0,C 180,E1 -15909.086,E2 -15909.086} C_VEL
LIN {X 0,Y 467.574,Z 492.572,A -85,B 0,C 180,E1 -15910.533,E2 -15910.533} C_VEL
LIN {X 0,Y 466.805,Z 507.153,A -85,B 0,C 180,E1 -15910.924,E2 -15910.924} C_VEL
LIN {X 0,Y 465.642,Z 521,A -85,B 0,C 180,E1 -15911.465,E2 -15911.465} C_VEL
LIN {X 0,Y 464.551,Z 533.281,A -85,B 0,C 180,E1 -15912.111,E2 -15912.111} C_VEL
LIN {X 0,Y 463.215,Z 546.048,A -85,B 0,C 180,E1 -15912.966,E2 -15912.966} C_VEL
LIN {X 0,Y 461.814,Z 557.68,A -85,B 0,C 180,E1 -15913.933,E2 -15913.933} C_VEL
LIN {X 0,Y 460.438,Z 568.372,A -85,B 0,C 180,E1 -15915.015,E2 -15915.015} C_VEL
LIN {X 0,Y 459.11,Z 578.993,A -85,B 0,C 180,E1 -15916.324,E2 -15916.324} C_VEL
LIN {X 0,Y 458.114,Z 587.795,A -85,B 0,C 180,E1 -15917.642,E2 -15917.642} C_VEL
LIN {X 0,Y 457.159,Z 596.307,A -85,B 0,C 180,E1 -15919.191,E2 -15919.191} C_VEL
LIN {X 0,Y 456.421,Z 603.132,A -85,B 0,C 180,E1 -15920.729,E2 -15920.729} C_VEL
LIN {X 0,Y 455.901,Z 609.304,A -85,B 0,C 180,E1 -15922.498,E2 -15922.498} C_VEL
LIN {X 0,Y 455.779,Z 612.987,A -85,B 0,C 180,E1 -15923.827,E2 -15923.827} C_VEL
LIN {X 0,Y 455.703,Z 617.317,A -85,B 0,C 180,E1 -15925.153,E2 -15925.153} C_VEL
LIN {X 0,Y 455.655,Z 620.707,A -85,B 0,C 180,E1 -15926.477,E2 -15926.477} C_VEL
LIN {X 0,Y 455.667,Z 622.969,A -85,B 0,C 180,E1 -15927.667,E2 -15927.667} C_VEL
LIN {X 0,Y 455.72,Z 624.796,A -85,B 0,C 180,E1 -15929.121,E2 -15929.121} C_VEL
LIN {X 0,Y 455.681,Z 625.673,A -85,B 0,C 180,E1 -15930.883,E2 -15930.883} C_VEL
LIN {X 0,Y 455.639,Z 625.097,A -85,B 0,C 180,E1 -15932.645,E2 -15932.645} C_VEL
LIN {X 0,Y 455.691,Z 623.074,A -85,B 0,C 180,E1 -15934.41,E2 -15934.41} C_VEL
LIN {X 0,Y 455.857,Z 619.537,A -85,B 0,C 180,E1 -15936.177,E2 -15936.177} C_VEL
LIN {X 0,Y 456.21,Z 614.42,A -85,B 0,C 180,E1 -15937.945,E2 -15937.945} C_VEL
LIN {X 0,Y 456.694,Z 609.486,A -85,B 0,C 180,E1 -15939.269,E2 -15939.269} C_VEL
LIN {X 0,Y 457.567,Z 602.336,A -85,B 0,C 180,E1 -15940.81,E2 -15940.81} C_VEL
LIN {X 0,Y 458.318,Z 594.833,A -85,B 0,C 180,E1 -15942.139,E2 -15942.139} C_VEL
LIN {X 0,Y 459.364,Z 585.918,A -85,B 0,C 180,E1 -15943.448,E2 -15943.448} C_VEL
LIN {X 0,Y 460.681,Z 575.119,A -85,B 0,C 180,E1 -15944.756,E2 -15944.756} C_VEL
LIN {X 0,Y 462.025,Z 563.093,A -85,B 0,C 180,E1 -15945.951,E2 -15945.951} C_VEL
LIN {X 0,Y 463.311,Z 551.057,A -85,B 0,C 180,E1 -15946.921,E2 -15946.921} C_VEL
LIN {X 0,Y 464.635,Z 537.819,A -85,B 0,C 180,E1 -15947.776,E2 -15947.776} C_VEL
LIN {X 0,Y 465.825,Z 524.04,A -85,B 0,C 180,E1 -15948.471,E2 -15948.471} C_VEL
LIN {X 0,Y 466.902,Z 509.341,A -85,B 0,C 180,E1 -15949.019,E2 -15949.019} C_VEL
LIN {X 0,Y 467.737,Z 493.538,A -85,B 0,C 180,E1 -15949.408,E2 -15949.408} C_VEL
LIN {X 0,Y 471.293,Z 402.234,A -85,B 0,C 180,E1 -15951.346,E2 -15951.346} C_VEL
LIN {X 0,Y 469.959,Z 386.107,A -85,B 0,C 180,E1 -15951.849,E2 -15951.849} C_VEL
LIN {X 0,Y 466.77,Z 363.275,A -85,B 0,C 180,E1 -15952.685,E2 -15952.685} C_VEL
LIN {X 0,Y 465.067,Z 353.535,A -85,B 0,C 180,E1 -15953.108,E2 -15953.108} C_VEL
LIN {X 0,Y 462.812,Z 332.725,A -85,B 0,C 180,E1 -15954.546,E2 -15954.546} C_VEL
LIN {X 0,Y 461.863,Z 322.732,A -85,B 0,C 180,E1 -15955.31,E2 -15955.31} C_VEL
LIN {X 0,Y 459.684,Z 310.113,A -85,B 0,C 180,E1 -15957.498,E2 -15957.498} C_VEL
LIN {X 0,Y 457.635,Z 300.041,A -85,B 0,C 180,E1 -15959.328,E2 -15959.328} C_VEL
LIN {X 0,Y 457.53,Z 300.045,A -85,B 0,C 180,E1 -15962.647,E2 -15962.647} C_VEL
LIN {X 0,Y 457.561,Z 300.049,A -85,B 0,C 180,E1 -15965.773,E2 -15965.773} C_VEL
LIN {X 0,Y 457.561,Z 300.048,A -85,B 0,C 180,E1 -15968.878,E2 -15968.878} C_VEL
LIN {X 0,Y 457.58,Z 300.041,A -85,B 0,C 180,E1 -15972.342,E2 -15972.342} C_VEL
LIN {X 0,Y 457.597,Z 300.041,A -85,B 0,C 180,E1 -15975.241,E2 -15975.241} C_VEL
LIN {X 0,Y 457.59,Z 300.042,A -85,B 0,C 180,E1 -15978.597,E2 -15978.597} C_VEL
LIN {X 0,Y 457.569,Z 300.046,A -85,B 0,C 180,E1 -15981.327,E2 -15981.327} C_VEL
LIN {X 0,Y 457.604,Z 300.041,A -85,B 0,C 180,E1 -15984.433,E2 -15984.433} C_VEL
LIN {X 0,Y 457.592,Z 300.042,A -85,B 0,C 180,E1 -15987.605,E2 -15987.605} C_VEL
LIN {X 0,Y 457.637,Z 300.04,A -85,B 0,C 180,E1 -15990.744,E2 -15990.744} C_VEL
LIN {X 0,Y 457.632,Z 300.04,A -85,B 0,C 180,E1 -15993.649,E2 -15993.649} C_VEL
LIN {X 0,Y 457.627,Z 300.047,A -85,B 0,C 180,E1 -15996.691,E2 -15996.691} C_VEL
LIN {X 0,Y 457.67,Z 300.043,A -85,B 0,C 180,E1 -15999.39,E2 -15999.39} C_VEL
LIN {X 0,Y 457.681,Z 300.251,A -85,B 0,C 180,E1 -16000.732,E2 -16000.732} C_VEL
LIN {X 0,Y 461.365,Z 311.328,A -85,B 0,C 180,E1 -16003.036,E2 -16003.036} C_VEL
LIN {X 0,Y 464.447,Z 322.193,A -85,B 0,C 180,E1 -16005.145,E2 -16005.145} C_VEL
LIN {X 0,Y 466.565,Z 332.478,A -85,B 0,C 180,E1 -16006.986,E2 -16006.986} C_VEL
LIN {X 0,Y 466.669,Z 335.806,A -85,B 0,C 180,E1 -16007.529,E2 -16007.529} C_VEL
LIN {X 0,Y 465.921,Z 345.76,A -85,B 0,C 180,E1 -16009.032,E2 -16009.032} C_VEL
LIN {X 0,Y 470.431,Z 365.89,A -85,B 0,C 180,E1 -16009.916,E2 -16009.916} C_VEL
LIN {X 0,Y 472.547,Z 377.886,A -85,B 0,C 180,E1 -16010.376,E2 -16010.376} C_VEL
LIN {X 0,Y 468.154,Z 485.853,A -85,B 0,C 180,E1 -16012.667,E2 -16012.667} C_VEL
LIN {X 0,Y 467.337,Z 499.668,A -85,B 0,C 180,E1 -16013.113,E2 -16013.113} C_VEL
LIN {X 0,Y 466.223,Z 514.755,A -85,B 0,C 180,E1 -16013.801,E2 -16013.801} C_VEL
LIN {X 0,Y 464.91,Z 528.597,A -85,B 0,C 180,E1 -16014.622,E2 -16014.622} C_VEL
LIN {X 0,Y 463.604,Z 541.251,A -85,B 0,C 180,E1 -16015.572,E2 -16015.572} C_VEL
LIN {X 0,Y 462.337,Z 552.695,A -85,B 0,C 180,E1 -16016.634,E2 -16016.634} C_VEL
LIN {X 0,Y 461.08,Z 563.299,A -85,B 0,C 180,E1 -16017.823,E2 -16017.823} C_VEL
LIN {X 0,Y 459.773,Z 572.953,A -85,B 0,C 180,E1 -16019.127,E2 -16019.127} C_VEL
LIN {X 0,Y 458.635,Z 581.001,A -85,B 0,C 180,E1 -16020.437,E2 -16020.437} C_VEL
LIN {X 0,Y 457.656,Z 588.704,A -85,B 0,C 180,E1 -16021.973,E2 -16021.973} C_VEL
LIN {X 0,Y 456.878,Z 594.886,A -85,B 0,C 180,E1 -16023.516,E2 -16023.516} C_VEL
LIN {X 0,Y 456.565,Z 599.065,A -85,B 0,C 180,E1 -16024.84,E2 -16024.84} C_VEL
LIN {X 0,Y 456.164,Z 602.397,A -85,B 0,C 180,E1 -16026.17,E2 -16026.17} C_VEL
LIN {X 0,Y 455.739,Z 605.468,A -85,B 0,C 180,E1 -16027.951,E2 -16027.951} C_VEL
LIN {X 0,Y 455.638,Z 607.07,A -85,B 0,C 180,E1 -16029.736,E2 -16029.736} C_VEL
LIN {X 0,Y 455.48,Z 607.23,A -85,B 0,C 180,E1 -16031.532,E2 -16031.532} C_VEL
LIN {X 0,Y 455.498,Z 605.907,A -85,B 0,C 180,E1 -16033.336,E2 -16033.336} C_VEL
LIN {X 0,Y 455.569,Z 604.41,A -85,B 0,C 180,E1 -16034.383,E2 -16034.383} C_VEL
LIN {X 0,Y 455.622,Z 600.937,A -85,B 0,C 180,E1 -16036.065,E2 -16036.065} C_VEL
LIN {X 0,Y 455.827,Z 596.224,A -85,B 0,C 180,E1 -16037.685,E2 -16037.685} C_VEL
LIN {X 0,Y 456.119,Z 590.15,A -85,B 0,C 180,E1 -16039.279,E2 -16039.279} C_VEL
LIN {X 0,Y 456.453,Z 583.54,A -85,B 0,C 180,E1 -16040.667,E2 -16040.667} C_VEL
LIN {X 0,Y 456.911,Z 575.483,A -85,B 0,C 180,E1 -16042.06,E2 -16042.06} C_VEL
LIN {X 0,Y 457.51,Z 565.679,A -85,B 0,C 180,E1 -16043.457,E2 -16043.457} C_VEL
LIN {X 0,Y 458.174,Z 554.644,A -85,B 0,C 180,E1 -16044.74,E2 -16044.74} C_VEL
LIN {X 0,Y 458.973,Z 542.095,A -85,B 0,C 180,E1 -16045.932,E2 -16045.932} C_VEL
LIN {X 0,Y 459.747,Z 528.812,A -85,B 0,C 180,E1 -16046.953,E2 -16046.953} C_VEL
LIN {X 0,Y 460.446,Z 515.361,A -85,B 0,C 180,E1 -16047.767,E2 -16047.767} C_VEL
LIN {X 0,Y 461.08,Z 501.799,A -85,B 0,C 180,E1 -16048.403,E2 -16048.403} C_VEL
LIN {X 0,Y 461.716,Z 486.668,A -85,B 0,C 180,E1 -16048.918,E2 -16048.918} C_VEL
LIN {X 0,Y 462.129,Z 467.757,A -85,B 0,C 180,E1 -16049.325,E2 -16049.325} C_VEL
LIN {X 0,Y 464.131,Z 373.105,A -85,B 0,C 180,E1 -16051.133,E2 -16051.133} C_VEL
LIN {X 0,Y 460.243,Z 343.81,A -85,B 0,C 180,E1 -16051.86,E2 -16051.86} C_VEL
LIN {X 0,Y 461.281,Z 322.319,A -85,B 0,C 180,E1 -16055.026,E2 -16055.026} C_VEL
LIN {X 0,Y 461.361,Z 319.124,A -85,B 0,C 180,E1 -16055.501,E2 -16055.501} C_VEL
LIN {X 0,Y 458.541,Z 304.621,A -85,B 0,C 180,E1 -16057.786,E2 -16057.786} C_VEL
LIN {X 0,Y 457.591,Z 300.046,A -85,B 0,C 180,E1 -16058.517,E2 -16058.517} C_VEL
LIN {X 0,Y 457.594,Z 300.038,A -85,B 0,C 180,E1 -16061.403,E2 -16061.403} C_VEL
LIN {X 0,Y 457.607,Z 300.04,A -85,B 0,C 180,E1 -16064.757,E2 -16064.757} C_VEL
LIN {X 0,Y 457.58,Z 300.041,A -85,B 0,C 180,E1 -16067.658,E2 -16067.658} C_VEL
LIN {X 0,Y 457.56,Z 300.043,A -85,B 0,C 180,E1 -16071.122,E2 -16071.122} C_VEL
LIN {X 0,Y 457.567,Z 300.047,A -85,B 0,C 180,E1 -16074.428,E2 -16074.428} C_VEL
LIN {X 0,Y 457.573,Z 300.043,A -85,B 0,C 180,E1 -16077.602,E2 -16077.602} C_VEL
LIN {X 0,Y 457.634,Z 300.035,A -85,B 0,C 180,E1 -16080.742,E2 -16080.742} C_VEL
LIN {X 0,Y 457.608,Z 300.04,A -85,B 0,C 180,E1 -16083.646,E2 -16083.646} C_VEL
LIN {X 0,Y 457.623,Z 300.036,A -85,B 0,C 180,E1 -16086.689,E2 -16086.689} C_VEL
LIN {X 0,Y 457.667,Z 300.031,A -85,B 0,C 180,E1 -16089.388,E2 -16089.388} C_VEL
LIN {X 0,Y 457.67,Z 300.034,A -85,B 0,C 180,E1 -16092.174,E2 -16092.174} C_VEL
LIN {X 0,Y 457.731,Z 300.021,A -85,B 0,C 180,E1 -16094.92,E2 -16094.92} C_VEL
LIN {X 0,Y 457.762,Z 300.018,A -85,B 0,C 180,E1 -16098.524,E2 -16098.524} C_VEL
LIN {X 0,Y 457.794,Z 300.106,A -85,B 0,C 180,E1 -16100.698,E2 -16100.698} C_VEL
LIN {X 0,Y 458.903,Z 306.037,A -85,B 0,C 180,E1 -16102.013,E2 -16102.013} C_VEL
LIN {X 0,Y 462.884,Z 319.532,A -85,B 0,C 180,E1 -16102.378,E2 -16102.378} C_VEL
LIN {X 0,Y 465.18,Z 331.772,A -85,B 0,C 180,E1 -16102.657,E2 -16102.657} C_VEL
LIN {X 0,Y 463.372,Z 441.72,A -85,B 0,C 180,E1 -16104.359,E2 -16104.359} C_VEL
LIN {X 0,Y 462.98,Z 456.138,A -85,B 0,C 180,E1 -16104.763,E2 -16104.763} C_VEL
LIN {X 0,Y 462.453,Z 469.951,A -85,B 0,C 180,E1 -16105.328,E2 -16105.328} C_VEL
LIN {X 0,Y 461.766,Z 483.69,A -85,B 0,C 180,E1 -16106.084,E2 -16106.084} C_VEL
LIN {X 0,Y 461.007,Z 496.019,A -85,B 0,C 180,E1 -16106.95,E2 -16106.95} C_VEL
LIN {X 0,Y 459.94,Z 508.516,A -85,B 0,C 180,E1 -16108.034,E2 -16108.034} C_VEL
LIN {X 0,Y 459.345,Z 518.656,A -85,B 0,C 180,E1 -16109.124,E2 -16109.124} C_VEL
LIN {X 0,Y 458.386,Z 528.835,A -85,B 0,C 180,E1 -16110.436,E2 -16110.436} C_VEL
LIN {X 0,Y 457.771,Z 537.234,A -85,B 0,C 180,E1 -16111.751,E2 -16111.751} C_VEL
LIN {X 0,Y 456.999,Z 545.294,A -85,B 0,C 180,E1 -16113.293,E2 -16113.293} C_VEL
LIN {X 0,Y 456.94,Z 547.525,A -85,B 0,C 180,E1 -16113.791,E2 -16113.791} C_VEL
LIN {X 0,Y 456.189,Z 550.321,A -85,B 0,C 180,E1 -16114.436,E2 -16114.436} C_VEL
LIN {X 0,Y 453.072,Z 554.48,A -85,B 0,C 180,E1 -16115.501,E2 -16115.501} C_VEL
LIN {X 0,Y 449.896,Z 558.032,A -85,B 0,C 180,E1 -16116.613,E2 -16116.613} C_VEL
LIN {X 0,Y 449.074,Z 559.88,A -85,B 0,C 180,E1 -16117.325,E2 -16117.325} C_VEL
LIN {X 0,Y 448.856,Z 563.23,A -85,B 0,C 180,E1 -16118.975,E2 -16118.975} C_VEL
LIN {X 0,Y 448.8,Z 565.554,A -85,B 0,C 180,E1 -16120.792,E2 -16120.792} C_VEL
LIN {X 0,Y 448.791,Z 566.529,A -85,B 0,C 180,E1 -16122.619,E2 -16122.619} C_VEL
LIN {X 0,Y 449.031,Z 566.146,A -85,B 0,C 180,E1 -16124.45,E2 -16124.45} C_VEL
LIN {X 0,Y 449.234,Z 564.402,A -85,B 0,C 180,E1 -16126.297,E2 -16126.297} C_VEL
LIN {X 0,Y 449.78,Z 561.082,A -85,B 0,C 180,E1 -16128.203,E2 -16128.203} C_VEL
LIN {X 0,Y 450.469,Z 556.422,A -85,B 0,C 180,E1 -16130.001,E2 -16130.001} C_VEL
LIN {X 0,Y 451.202,Z 551.395,A -85,B 0,C 180,E1 -16131.485,E2 -16131.485} C_VEL
LIN {X 0,Y 452.146,Z 544.855,A -85,B 0,C 180,E1 -16133.024,E2 -16133.024} C_VEL
LIN {X 0,Y 453.157,Z 538.13,A -85,B 0,C 180,E1 -16134.322,E2 -16134.322} C_VEL
LIN {X 0,Y 454.473,Z 528.753,A -85,B 0,C 180,E1 -16135.808,E2 -16135.808} C_VEL
LIN {X 0,Y 455.879,Z 518.692,A -85,B 0,C 180,E1 -16137.106,E2 -16137.106} C_VEL
LIN {X 0,Y 457.136,Z 508.16,A -85,B 0,C 180,E1 -16138.232,E2 -16138.232} C_VEL
LIN {X 0,Y 458.452,Z 496.301,A -85,B 0,C 180,E1 -16139.266,E2 -16139.266} C_VEL
LIN {X 0,Y 459.667,Z 483.138,A -85,B 0,C 180,E1 -16140.186,E2 -16140.186} C_VEL
LIN {X 0,Y 460.542,Z 470.471,A -85,B 0,C 180,E1 -16140.881,E2 -16140.881} C_VEL
LIN {X 0,Y 461.405,Z 456.65,A -85,B 0,C 180,E1 -16141.444,E2 -16141.444} C_VEL
LIN {X 0,Y 461.865,Z 442.947,A -85,B 0,C 180,E1 -16141.834,E2 -16141.834} C_VEL
LIN {X 0,Y 462.949,Z 384.93,A -85,B 0,C 180,E1 -16142.774,E2 -16142.774} C_VEL
LIN {X 0,Y 464.029,Z 335.954,A -85,B 0,C 180,E1 -16143.538,E2 -16143.538} C_VEL
LIN {X 0,Y 457.042,Z 318.916,A -85,B 0,C 180,E1 -16144.253,E2 -16144.253} C_VEL
LIN {X 0,Y 452.02,Z 307.541,A -85,B 0,C 180,E1 -16144.787,E2 -16144.787} C_VEL
LIN {X 0,Y 450.514,Z 300.928,A -85,B 0,C 180,E1 -16146.488,E2 -16146.488} C_VEL
LIN {X 0,Y 450.486,Z 300.927,A -85,B 0,C 180,E1 -16149.602,E2 -16149.602} C_VEL
LIN {X 0,Y 450.525,Z 300.917,A -85,B 0,C 180,E1 -16151.95,E2 -16151.95} C_VEL
LIN {X 0,Y 450.541,Z 300.909,A -85,B 0,C 180,E1 -16154.391,E2 -16154.391} C_VEL
LIN {X 0,Y 450.53,Z 300.922,A -85,B 0,C 180,E1 -16156.942,E2 -16156.942} C_VEL
LIN {X 0,Y 450.51,Z 300.923,A -85,B 0,C 180,E1 -16160.397,E2 -16160.397} C_VEL
LIN {X 0,Y 450.528,Z 300.9,A -85,B 0,C 180,E1 -16163.787,E2 -16163.787} C_VEL
LIN {X 0,Y 450.535,Z 300.92,A -85,B 0,C 180,E1 -16167.086,E2 -16167.086} C_VEL
LIN {X 0,Y 450.538,Z 300.922,A -85,B 0,C 180,E1 -16170.165,E2 -16170.165} C_VEL
LIN {X 0,Y 450.57,Z 300.909,A -85,B 0,C 180,E1 -16173.203,E2 -16173.203} C_VEL
LIN {X 0,Y 450.559,Z 300.908,A -85,B 0,C 180,E1 -16176.515,E2 -16176.515} C_VEL
LIN {X 0,Y 450.571,Z 300.911,A -85,B 0,C 180,E1 -16180.001,E2 -16180.001} C_VEL
LIN {X 0,Y 450.563,Z 300.915,A -85,B 0,C 180,E1 -16182.82,E2 -16182.82} C_VEL
LIN {X 0,Y 450.614,Z 300.901,A -85,B 0,C 180,E1 -16185.599,E2 -16185.599} C_VEL
LIN {X 0,Y 450.707,Z 300.898,A -85,B 0,C 180,E1 -16188.344,E2 -16188.344} C_VEL
LIN {X 0,Y 450.756,Z 300.888,A -85,B 0,C 180,E1 -16191.961,E2 -16191.961} C_VEL
LIN {X 0,Y 450.792,Z 300.889,A -85,B 0,C 180,E1 -16194.651,E2 -16194.651} C_VEL
LIN {X 0,Y 450.702,Z 300.893,A -85,B 0,C 180,E1 -16197.328,E2 -16197.328} C_VEL
LIN {X 0,Y 450.85,Z 300.878,A -85,B 0,C 180,E1 -16200,E2 -16200} C_VEL
LIN {X 0,Y 450.854,Z 300.88,A -85,B 0,C 180,E1 -16204.455,E2 -16204.455} C_VEL
LIN {X 0,Y 450.751,Z 300.881,A -85,B 0,C 180,E1 -16207.141,E2 -16207.141} C_VEL
LIN {X 0,Y 450.743,Z 300.894,A -85,B 0,C 180,E1 -16210.747,E2 -16210.747} C_VEL
LIN {X 0,Y 450.649,Z 300.9,A -85,B 0,C 180,E1 -16213.482,E2 -16213.482} C_VEL
LIN {X 0,Y 450.603,Z 300.909,A -85,B 0,C 180,E1 -16216.248,E2 -16216.248} C_VEL
LIN {X 0,Y 450.571,Z 300.916,A -85,B 0,C 180,E1 -16219.054,E2 -16219.054} C_VEL
LIN {X 0,Y 450.556,Z 300.909,A -85,B 0,C 180,E1 -16221.908,E2 -16221.908} C_VEL
LIN {X 0,Y 450.513,Z 300.924,A -85,B 0,C 180,E1 -16224.821,E2 -16224.821} C_VEL
LIN {X 0,Y 450.56,Z 300.915,A -85,B 0,C 180,E1 -16227.8,E2 -16227.8} C_VEL
LIN {X 0,Y 450.578,Z 300.912,A -85,B 0,C 180,E1 -16230.864,E2 -16230.864} C_VEL
LIN {X 0,Y 450.553,Z 300.908,A -85,B 0,C 180,E1 -16234.033,E2 -16234.033} C_VEL
LIN {X 0,Y 450.587,Z 300.906,A -85,B 0,C 180,E1 -16237.32,E2 -16237.32} C_VEL
LIN {X 0,Y 450.553,Z 300.917,A -85,B 0,C 180,E1 -16240.384,E2 -16240.384} C_VEL
LIN {X 0,Y 450.555,Z 300.916,A -85,B 0,C 180,E1 -16243.16,E2 -16243.16} C_VEL
LIN {X 0,Y 450.56,Z 300.915,A -85,B 0,C 180,E1 -16245.653,E2 -16245.653} C_VEL
LIN {X 0,Y 450.574,Z 300.92,A -85,B 0,C 180,E1 -16248.261,E2 -16248.261} C_VEL
LIN {X 0,Y 450.573,Z 300.917,A -85,B 0,C 180,E1 -16251.554,E2 -16251.554} C_VEL
LIN {X 0,Y 450.584,Z 300.923,A -85,B 0,C 180,E1 -16254.891,E2 -16254.891} C_VEL
LIN {X 0,Y 450.596,Z 301.081,A -85,B 0,C 180,E1 -16257.541,E2 -16257.541} C_VEL
LIN {X 0,Y 453.968,Z 314.872,A -85,B 0,C 180,E1 -16260.416,E2 -16260.416} C_VEL
LIN {X 0,Y 456.597,Z 327.193,A -85,B 0,C 180,E1 -16262.842,E2 -16262.842} C_VEL
LIN {X 0,Y 457.396,Z 331.347,A -85,B 0,C 180,E1 -16263.637,E2 -16263.637} C_VEL
LIN {X 0,Y 456.089,Z 343.742,A -85,B 0,C 180,E1 -16265.747,E2 -16265.747} C_VEL
LIN {X 0,Y 454.928,Z 353.969,A -85,B 0,C 180,E1 -16267.46,E2 -16267.46} C_VEL
LIN {X 0,Y 459.748,Z 380.25,A -85,B 0,C 180,E1 -16268.206,E2 -16268.206} C_VEL
LIN {X 0,Y 462.782,Z 401.053,A -85,B 0,C 180,E1 -16268.732,E2 -16268.732} C_VEL
LIN {X 0,Y 461.047,Z 492.239,A -85,B 0,C 180,E1 -16270.188,E2 -16270.188} C_VEL
LIN {X 0,Y 460.22,Z 506.848,A -85,B 0,C 180,E1 -16270.585,E2 -16270.585} C_VEL
LIN {X 0,Y 459.03,Z 520.794,A -85,B 0,C 180,E1 -16271.14,E2 -16271.14} C_VEL
LIN {X 0,Y 457.827,Z 533.768,A -85,B 0,C 180,E1 -16271.839,E2 -16271.839} C_VEL
LIN {X 0,Y 456.461,Z 546.36,A -85,B 0,C 180,E1 -16272.706,E2 -16272.706} C_VEL
LIN {X 0,Y 455.016,Z 557.863,A -85,B 0,C 180,E1 -16273.686,E2 -16273.686} C_VEL
LIN {X 0,Y 453.562,Z 568.447,A -85,B 0,C 180,E1 -16274.782,E2 -16274.782} C_VEL
LIN {X 0,Y 452.207,Z 578.979,A -85,B 0,C 180,E1 -16276.111,E2 -16276.111} C_VEL
LIN {X 0,Y 451.156,Z 587.708,A -85,B 0,C 180,E1 -16277.449,E2 -16277.449} C_VEL
LIN {X 0,Y 450.201,Z 595.711,A -85,B 0,C 180,E1 -16278.932,E2 -16278.932} C_VEL
LIN {X 0,Y 449.387,Z 602.931,A -85,B 0,C 180,E1 -16280.583,E2 -16280.583} C_VEL
LIN {X 0,Y 448.813,Z 609.034,A -85,B 0,C 180,E1 -16282.379,E2 -16282.379} C_VEL
LIN {X 0,Y 448.701,Z 612.537,A -85,B 0,C 180,E1 -16283.729,E2 -16283.729} C_VEL
LIN {X 0,Y 448.603,Z 618.141,A -85,B 0,C 180,E1 -16285.525,E2 -16285.525} C_VEL
LIN {X 0,Y 448.584,Z 620.336,A -85,B 0,C 180,E1 -16286.421,E2 -16286.421} C_VEL
LIN {X 0,Y 448.592,Z 623.52,A -85,B 0,C 180,E1 -16288.213,E2 -16288.213} C_VEL
LIN {X 0,Y 448.631,Z 624.547,A -85,B 0,C 180,E1 -16289.108,E2 -16289.108} C_VEL
LIN {X 0,Y 448.595,Z 625.499,A -85,B 0,C 180,E1 -16290.897,E2 -16290.897} C_VEL
LIN {X 0,Y 448.545,Z 625,A -85,B 0,C 180,E1 -16292.687,E2 -16292.687} C_VEL
LIN {X 0,Y 448.6,Z 623.059,A -85,B 0,C 180,E1 -16294.48,E2 -16294.48} C_VEL
LIN {X 0,Y 448.774,Z 619.631,A -85,B 0,C 180,E1 -16296.274,E2 -16296.274} C_VEL
LIN {X 0,Y 449.154,Z 614.608,A -85,B 0,C 180,E1 -16298.07,E2 -16298.07} C_VEL
LIN {X 0,Y 449.695,Z 609.755,A -85,B 0,C 180,E1 -16299.415,E2 -16299.415} C_VEL
LIN {X 0,Y 450.605,Z 602.702,A -85,B 0,C 180,E1 -16300.979,E2 -16300.979} C_VEL
LIN {X 0,Y 451.384,Z 595.576,A -85,B 0,C 180,E1 -16302.287,E2 -16302.287} C_VEL
LIN {X 0,Y 452.488,Z 586.541,A -85,B 0,C 180,E1 -16303.657,E2 -16303.657} C_VEL
LIN {X 0,Y 453.882,Z 575.894,A -85,B 0,C 180,E1 -16304.983,E2 -16304.983} C_VEL
LIN {X 0,Y 455.273,Z 564.092,A -85,B 0,C 180,E1 -16306.194,E2 -16306.194} C_VEL
LIN {X 0,Y 456.772,Z 550.908,A -85,B 0,C 180,E1 -16307.286,E2 -16307.286} C_VEL
LIN {X 0,Y 458.197,Z 537.686,A -85,B 0,C 180,E1 -16308.15,E2 -16308.15} C_VEL
LIN {X 0,Y 459.357,Z 524.721,A -85,B 0,C 180,E1 -16308.822,E2 -16308.822} C_VEL
LIN {X 0,Y 460.542,Z 509.527,A -85,B 0,C 180,E1 -16309.406,E2 -16309.406} C_VEL
LIN {X 0,Y 461.424,Z 494.183,A -85,B 0,C 180,E1 -16309.797,E2 -16309.797} C_VEL
LIN {X 0,Y 465.167,Z 403.031,A -85,B 0,C 180,E1 -16311.778,E2 -16311.778} C_VEL
LIN {X 0,Y 464.003,Z 388.072,A -85,B 0,C 180,E1 -16312.256,E2 -16312.256} C_VEL
LIN {X 0,Y 461.12,Z 366.645,A -85,B 0,C 180,E1 -16313.061,E2 -16313.061} C_VEL
LIN {X 0,Y 458.907,Z 354.217,A -85,B 0,C 180,E1 -16313.596,E2 -16313.596} C_VEL
LIN {X 0,Y 457.249,Z 336.764,A -85,B 0,C 180,E1 -16314.827,E2 -16314.827} C_VEL
LIN {X 0,Y 456.042,Z 325.449,A -85,B 0,C 180,E1 -16315.717,E2 -16315.717} C_VEL
LIN {X 0,Y 453.766,Z 317.051,A -85,B 0,C 180,E1 -16316.595,E2 -16316.595} C_VEL
LIN {X 0,Y 450.936,Z 302.5,A -85,B 0,C 180,E1 -16319.217,E2 -16319.217} C_VEL
LIN {X 0,Y 450.581,Z 300.916,A -85,B 0,C 180,E1 -16319.518,E2 -16319.518} C_VEL
LIN {X 0,Y 450.502,Z 300.922,A -85,B 0,C 180,E1 -16322.971,E2 -16322.971} C_VEL
LIN {X 0,Y 450.517,Z 300.926,A -85,B 0,C 180,E1 -16326.216,E2 -16326.216} C_VEL
LIN {X 0,Y 450.505,Z 300.926,A -85,B 0,C 180,E1 -16329.605,E2 -16329.605} C_VEL
LIN {X 0,Y 450.533,Z 300.92,A -85,B 0,C 180,E1 -16331.955,E2 -16331.955} C_VEL
LIN {X 0,Y 450.563,Z 300.917,A -85,B 0,C 180,E1 -16334.395,E2 -16334.395} C_VEL
LIN {X 0,Y 450.541,Z 300.92,A -85,B 0,C 180,E1 -16336.947,E2 -16336.947} C_VEL
LIN {X 0,Y 450.517,Z 300.923,A -85,B 0,C 180,E1 -16339.628,E2 -16339.628} C_VEL
LIN {X 0,Y 450.515,Z 300.926,A -85,B 0,C 180,E1 -16342.673,E2 -16342.673} C_VEL
LIN {X 0,Y 450.552,Z 300.918,A -85,B 0,C 180,E1 -16345.967,E2 -16345.967} C_VEL
LIN {X 0,Y 450.553,Z 300.921,A -85,B 0,C 180,E1 -16349.134,E2 -16349.134} C_VEL
LIN {X 0,Y 450.591,Z 300.917,A -85,B 0,C 180,E1 -16352.386,E2 -16352.386} C_VEL
LIN {X 0,Y 450.539,Z 300.925,A -85,B 0,C 180,E1 -16355.18,E2 -16355.18} C_VEL
LIN {X 0,Y 450.587,Z 300.925,A -85,B 0,C 180,E1 -16358.094,E2 -16358.094} C_VEL
LIN {X 0,Y 450.621,Z 300.959,A -85,B 0,C 180,E1 -16359.944,E2 -16359.944} C_VEL
LIN {X 0,Y 454.621,Z 312.732,A -85,B 0,C 180,E1 -16362.516,E2 -16362.516} C_VEL
LIN {X 0,Y 458.105,Z 324.959,A -85,B 0,C 180,E1 -16364.934,E2 -16364.934} C_VEL
LIN {X 0,Y 460.227,Z 335.794,A -85,B 0,C 180,E1 -16366.924,E2 -16366.924} C_VEL
LIN {X 0,Y 459.599,Z 345.911,A -85,B 0,C 180,E1 -16368.489,E2 -16368.489} C_VEL
LIN {X 0,Y 463.725,Z 363.93,A -85,B 0,C 180,E1 -16369.332,E2 -16369.332} C_VEL
LIN {X 0,Y 466.477,Z 378.734,A -85,B 0,C 180,E1 -16369.936,E2 -16369.936} C_VEL
LIN {X 0,Y 461.796,Z 486.961,A -85,B 0,C 180,E1 -16372.291,E2 -16372.291} C_VEL
LIN {X 0,Y 460.947,Z 500.43,A -85,B 0,C 180,E1 -16372.743,E2 -16372.743} C_VEL
LIN {X 0,Y 459.778,Z 515.335,A -85,B 0,C 180,E1 -16373.439,E2 -16373.439} C_VEL
LIN {X 0,Y 458.52,Z 527.872,A -85,B 0,C 180,E1 -16374.191,E2 -16374.191} C_VEL
LIN {X 0,Y 457.118,Z 540.858,A -85,B 0,C 180,E1 -16375.17,E2 -16375.17} C_VEL
LIN {X 0,Y 455.778,Z 552.521,A -85,B 0,C 180,E1 -16376.255,E2 -16376.255} C_VEL
LIN {X 0,Y 454.338,Z 564.021,A -85,B 0,C 180,E1 -16377.57,E2 -16377.57} C_VEL
LIN {X 0,Y 452.957,Z 573.576,A -85,B 0,C 180,E1 -16378.892,E2 -16378.892} C_VEL
LIN {X 0,Y 451.758,Z 581.56,A -85,B 0,C 180,E1 -16380.222,E2 -16380.222} C_VEL
LIN {X 0,Y 450.711,Z 589.192,A -85,B 0,C 180,E1 -16381.781,E2 -16381.781} C_VEL
LIN {X 0,Y 450.001,Z 594.496,A -85,B 0,C 180,E1 -16383.123,E2 -16383.123} C_VEL
LIN {X 0,Y 449.619,Z 598.805,A -85,B 0,C 180,E1 -16384.467,E2 -16384.467} C_VEL
LIN {X 0,Y 449.071,Z 603.153,A -85,B 0,C 180,E1 -16386.268,E2 -16386.268} C_VEL
LIN {X 0,Y 448.641,Z 605.999,A -85,B 0,C 180,E1 -16388.078,E2 -16388.078} C_VEL
LIN {X 0,Y 448.547,Z 607.381,A -85,B 0,C 180,E1 -16389.891,E2 -16389.891} C_VEL
LIN {X 0,Y 448.465,Z 607.523,A -85,B 0,C 180,E1 -16390.802,E2 -16390.802} C_VEL
LIN {X 0,Y 448.343,Z 606.661,A -85,B 0,C 180,E1 -16392.634,E2 -16392.634} C_VEL
LIN {X 0,Y 448.475,Z 604.292,A -85,B 0,C 180,E1 -16394.471,E2 -16394.471} C_VEL
LIN {X 0,Y 448.56,Z 600.334,A -85,B 0,C 180,E1 -16396.324,E2 -16396.324} C_VEL
LIN {X 0,Y 448.76,Z 595.934,A -85,B 0,C 180,E1 -16397.799,E2 -16397.799} C_VEL
LIN {X 0,Y 448.979,Z 590.958,A -85,B 0,C 180,E1 -16399.124,E2 -16399.124} C_VEL
LIN {X 0,Y 449.386,Z 583.462,A -85,B 0,C 180,E1 -16400.736,E2 -16400.736} C_VEL
LIN {X 0,Y 449.861,Z 575.144,A -85,B 0,C 180,E1 -16402.184,E2 -16402.184} C_VEL
LIN {X 0,Y 450.476,Z 565.316,A -85,B 0,C 180,E1 -16403.586,E2 -16403.586} C_VEL
LIN {X 0,Y 451.192,Z 554.025,A -85,B 0,C 180,E1 -16404.904,E2 -16404.904} C_VEL
LIN {X 0,Y 451.94,Z 542.182,A -85,B 0,C 180,E1 -16406.038,E2 -16406.038} C_VEL
LIN {X 0,Y 452.686,Z 529.458,A -85,B 0,C 180,E1 -16407.034,E2 -16407.034} C_VEL
LIN {X 0,Y 453.392,Z 516.268,A -85,B 0,C 180,E1 -16407.856,E2 -16407.856} C_VEL
LIN {X 0,Y 454.052,Z 503.093,A -85,B 0,C 180,E1 -16408.495,E2 -16408.495} C_VEL
LIN {X 0,Y 454.694,Z 488.061,A -85,B 0,C 180,E1 -16409.029,E2 -16409.029} C_VEL
LIN {X 0,Y 455.093,Z 471.477,A -85,B 0,C 180,E1 -16409.411,E2 -16409.411} C_VEL
LIN {X 0,Y 457.202,Z 373.391,A -85,B 0,C 180,E1 -16411.332,E2 -16411.332} C_VEL
LIN {X 0,Y 453.291,Z 343.834,A -85,B 0,C 180,E1 -16412.088,E2 -16412.088} C_VEL
LIN {X 0,Y 454.333,Z 322.894,A -85,B 0,C 180,E1 -16415.202,E2 -16415.202} C_VEL
LIN {X 0,Y 454.078,Z 318.418,A -85,B 0,C 180,E1 -16415.886,E2 -16415.886} C_VEL
LIN {X 0,Y 450.552,Z 300.921,A -85,B 0,C 180,E1 -16418.697,E2 -16418.697} C_VEL
LIN {X 0,Y 450.548,Z 300.919,A -85,B 0,C 180,E1 -16421.951,E2 -16421.951} C_VEL
LIN {X 0,Y 450.562,Z 300.922,A -85,B 0,C 180,E1 -16424.393,E2 -16424.393} C_VEL
LIN {X 0,Y 450.522,Z 300.921,A -85,B 0,C 180,E1 -16426.947,E2 -16426.947} C_VEL
LIN {X 0,Y 450.516,Z 300.921,A -85,B 0,C 180,E1 -16429.626,E2 -16429.626} C_VEL
LIN {X 0,Y 450.485,Z 300.927,A -85,B 0,C 180,E1 -16432.668,E2 -16432.668} C_VEL
LIN {X 0,Y 450.536,Z 300.923,A -85,B 0,C 180,E1 -16435.964,E2 -16435.964} C_VEL
LIN {X 0,Y 450.524,Z 300.919,A -85,B 0,C 180,E1 -16439.13,E2 -16439.13} C_VEL
LIN {X 0,Y 450.554,Z 300.915,A -85,B 0,C 180,E1 -16441.186,E2 -16441.186} C_VEL
LIN {X 0,Y 450.546,Z 300.92,A -85,B 0,C 180,E1 -16444.383,E2 -16444.383} C_VEL
LIN {X 0,Y 450.562,Z 300.914,A -85,B 0,C 180,E1 -16447.127,E2 -16447.127} C_VEL
LIN {X 0,Y 450.6,Z 300.917,A -85,B 0,C 180,E1 -16450,E2 -16450} C_VEL
LIN {X 0,Y 450.613,Z 300.908,A -85,B 0,C 180,E1 -16452.82,E2 -16452.82} C_VEL
LIN {X 0,Y 450.642,Z 300.908,A -85,B 0,C 180,E1 -16455.598,E2 -16455.598} C_VEL
LIN {X 0,Y 450.753,Z 300.893,A -85,B 0,C 180,E1 -16458.343,E2 -16458.343} C_VEL
LIN {X 0,Y 450.758,Z 300.989,A -85,B 0,C 180,E1 -16460.523,E2 -16460.523} C_VEL
LIN {X 0,Y 451.785,Z 306.456,A -85,B 0,C 180,E1 -16461.747,E2 -16461.747} C_VEL
LIN {X 0,Y 456.201,Z 320.991,A -85,B 0,C 180,E1 -16462.153,E2 -16462.153} C_VEL
LIN {X 0,Y 458.367,Z 332.986,A -85,B 0,C 180,E1 -16462.428,E2 -16462.428} C_VEL
LIN {X 0,Y 456.514,Z 441.86,A -85,B 0,C 180,E1 -16464.136,E2 -16464.136} C_VEL
LIN {X 0,Y 456.114,Z 456.377,A -85,B 0,C 180,E1 -16464.545,E2 -16464.545} C_VEL
LIN {X 0,Y 455.601,Z 469.679,A -85,B 0,C 180,E1 -16465.092,E2 -16465.092} C_VEL
LIN {X 0,Y 454.931,Z 482.702,A -85,B 0,C 180,E1 -16465.804,E2 -16465.804} C_VEL
LIN {X 0,Y 454.21,Z 495.285,A -85,B 0,C 180,E1 -16466.683,E2 -16466.683} C_VEL
LIN {X 0,Y 453.131,Z 506.841,A -85,B 0,C 180,E1 -16467.672,E2 -16467.672} C_VEL
LIN {X 0,Y 452.508,Z 516.384,A -85,B 0,C 180,E1 -16468.667,E2 -16468.667} C_VEL
LIN {X 0,Y 451.742,Z 525.399,A -85,B 0,C 180,E1 -16469.776,E2 -16469.776} C_VEL
LIN {X 0,Y 450.903,Z 534.463,A -85,B 0,C 180,E1 -16471.11,E2 -16471.11} C_VEL
LIN {X 0,Y 450.329,Z 542.002,A -85,B 0,C 180,E1 -16472.449,E2 -16472.449} C_VEL
LIN {X 0,Y 449.873,Z 548.038,A -85,B 0,C 180,E1 -16473.741,E2 -16473.741} C_VEL
LIN {X 0,Y 449.622,Z 552.659,A -85,B 0,C 180,E1 -16474.913,E2 -16474.913} C_VEL
LIN {X 0,Y 449.224,Z 558.324,A -85,B 0,C 180,E1 -16476.713,E2 -16476.713} C_VEL
LIN {X 0,Y 449.074,Z 559.88,A -85,B 0,C 180,E1 -16477.325,E2 -16477.325} C_VEL
LIN {X 0,Y 448.298,Z 561.545,A -85,B 0,C 180,E1 -16478.042,E2 -16478.042} C_VEL
LIN {X 0,Y 445.321,Z 563.862,A -85,B 0,C 180,E1 -16479.218,E2 -16479.218} C_VEL
LIN {X 0,Y 442.85,Z 565.284,A -85,B 0,C 180,E1 -16480.178,E2 -16480.178} C_VEL
LIN {X 0,Y 441.783,Z 566.052,A -85,B 0,C 180,E1 -16480.927,E2 -16480.927} C_VEL
LIN {X 0,Y 441.691,Z 566.233,A -85,B 0,C 180,E1 -16481.182,E2 -16481.182} C_VEL
LIN {X 0,Y 441.717,Z 566.972,A -85,B 0,C 180,E1 -16482.824,E2 -16482.824} C_VEL
LIN {X 0,Y 441.967,Z 566.495,A -85,B 0,C 180,E1 -16484.687,E2 -16484.687} C_VEL
LIN {X 0,Y 442.224,Z 564.645,A -85,B 0,C 180,E1 -16486.563,E2 -16486.563} C_VEL
LIN {X 0,Y 442.78,Z 561.314,A -85,B 0,C 180,E1 -16488.442,E2 -16488.442} C_VEL
LIN {X 0,Y 443.552,Z 556.412,A -85,B 0,C 180,E1 -16490.327,E2 -16490.327} C_VEL
LIN {X 0,Y 444.273,Z 551.61,A -85,B 0,C 180,E1 -16491.747,E2 -16491.747} C_VEL
LIN {X 0,Y 445.383,Z 544.597,A -85,B 0,C 180,E1 -16493.394,E2 -16493.394} C_VEL
LIN {X 0,Y 446.591,Z 536.911,A -85,B 0,C 180,E1 -16494.852,E2 -16494.852} C_VEL
LIN {X 0,Y 447.834,Z 528.18,A -85,B 0,C 180,E1 -16496.219,E2 -16496.219} C_VEL
LIN {X 0,Y 449.177,Z 518.871,A -85,B 0,C 180,E1 -16497.425,E2 -16497.425} C_VEL
LIN {X 0,Y 450.674,Z 507.149,A -85,B 0,C 180,E1 -16498.674,E2 -16498.674} C_VEL
LIN {X 0,Y 452.027,Z 494.975,A -85,B 0,C 180,E1 -16499.723,E2 -16499.723} C_VEL
LIN {X 0,Y 453.133,Z 483.222,A -85,B 0,C 180,E1 -16500.539,E2 -16500.539} C_VEL
LIN {X 0,Y 454.042,Z 470.458,A -85,B 0,C 180,E1 -16501.244,E2 -16501.244} C_VEL
LIN {X 0,Y 454.874,Z 456.515,A -85,B 0,C 180,E1 -16501.816,E2 -16501.816} C_VEL
LIN {X 0,Y 455.391,Z 443.211,A -85,B 0,C 180,E1 -16502.191,E2 -16502.191} C_VEL
LIN {X 0,Y 456.517,Z 385.369,A -85,B 0,C 180,E1 -16503.14,E2 -16503.14} C_VEL
LIN {X 0,Y 457.554,Z 337.663,A -85,B 0,C 180,E1 -16503.898,E2 -16503.898} C_VEL
LIN {X 0,Y 451.206,Z 322.138,A -85,B 0,C 180,E1 -16504.566,E2 -16504.566} C_VEL
LIN {X 0,Y 444.894,Z 308.02,A -85,B 0,C 180,E1 -16505.241,E2 -16505.241} C_VEL
LIN {X 0,Y 443.449,Z 301.806,A -85,B 0,C 180,E1 -16506.883,E2 -16506.883} C_VEL
LIN {X 0,Y 443.45,Z 301.801,A -85,B 0,C 180,E1 -16509.288,E2 -16509.288} C_VEL
LIN {X 0,Y 443.478,Z 301.804,A -85,B 0,C 180,E1 -16512.774,E2 -16512.774} C_VEL
LIN {X 0,Y 443.483,Z 301.793,A -85,B 0,C 180,E1 -16515.977,E2 -16515.977} C_VEL
LIN {X 0,Y 443.466,Z 301.803,A -85,B 0,C 180,E1 -16519.297,E2 -16519.297} C_VEL
LIN {X 0,Y 443.477,Z 301.799,A -85,B 0,C 180,E1 -16522.154,E2 -16522.154} C_VEL
LIN {X 0,Y 443.495,Z 301.779,A -85,B 0,C 180,E1 -16525.349,E2 -16525.349} C_VEL
LIN {X 0,Y 443.516,Z 301.79,A -85,B 0,C 180,E1 -16528.589,E2 -16528.589} C_VEL
LIN {X 0,Y 443.502,Z 301.795,A -85,B 0,C 180,E1 -16531.718,E2 -16531.718} C_VEL
LIN {X 0,Y 443.471,Z 301.8,A -85,B 0,C 180,E1 -16534.757,E2 -16534.757} C_VEL
LIN {X 0,Y 443.488,Z 301.796,A -85,B 0,C 180,E1 -16537.725,E2 -16537.725} C_VEL
LIN {X 0,Y 443.535,Z 301.786,A -85,B 0,C 180,E1 -16540.632,E2 -16540.632} C_VEL
LIN {X 0,Y 443.533,Z 301.798,A -85,B 0,C 180,E1 -16543.485,E2 -16543.485} C_VEL
LIN {X 0,Y 443.577,Z 301.777,A -85,B 0,C 180,E1 -16546.299,E2 -16546.299} C_VEL
LIN {X 0,Y 443.634,Z 301.784,A -85,B 0,C 180,E1 -16549.078,E2 -16549.078} C_VEL
LIN {X 0,Y 443.725,Z 301.765,A -85,B 0,C 180,E1 -16552.745,E2 -16552.745} C_VEL
LIN {X 0,Y 443.815,Z 301.748,A -85,B 0,C 180,E1 -16555.474,E2 -16555.474} C_VEL
LIN {X 0,Y 443.745,Z 301.771,A -85,B 0,C 180,E1 -16559.096,E2 -16559.096} C_VEL
LIN {X 0,Y 443.735,Z 301.76,A -85,B 0,C 180,E1 -16560.904,E2 -16560.904} C_VEL
LIN {X 0,Y 443.824,Z 301.756,A -85,B 0,C 180,E1 -16564.526,E2 -16564.526} C_VEL
LIN {X 0,Y 443.726,Z 301.755,A -85,B 0,C 180,E1 -16567.255,E2 -16567.255} C_VEL
LIN {X 0,Y 443.699,Z 301.769,A -85,B 0,C 180,E1 -16570.92,E2 -16570.92} C_VEL
LIN {X 0,Y 443.593,Z 301.778,A -85,B 0,C 180,E1 -16573.701,E2 -16573.701} C_VEL
LIN {X 0,Y 443.565,Z 301.783,A -85,B 0,C 180,E1 -16576.514,E2 -16576.514} C_VEL
LIN {X 0,Y 443.541,Z 301.79,A -85,B 0,C 180,E1 -16579.368,E2 -16579.368} C_VEL
LIN {X 0,Y 443.488,Z 301.788,A -85,B 0,C 180,E1 -16582.275,E2 -16582.275} C_VEL
LIN {X 0,Y 443.471,Z 301.797,A -85,B 0,C 180,E1 -16585.243,E2 -16585.243} C_VEL
LIN {X 0,Y 443.504,Z 301.798,A -85,B 0,C 180,E1 -16588.281,E2 -16588.281} C_VEL
LIN {X 0,Y 443.529,Z 301.791,A -85,B 0,C 180,E1 -16591.489,E2 -16591.489} C_VEL
LIN {X 0,Y 443.538,Z 301.768,A -85,B 0,C 180,E1 -16594.801,E2 -16594.801} C_VEL
LIN {X 0,Y 443.555,Z 301.786,A -85,B 0,C 180,E1 -16598.015,E2 -16598.015} C_VEL
LIN {X 0,Y 443.497,Z 301.797,A -85,B 0,C 180,E1 -16600.708,E2 -16600.708} C_VEL
LIN {X 0,Y 443.503,Z 301.799,A -85,B 0,C 180,E1 -16604.02,E2 -16604.02} C_VEL
LIN {X 0,Y 443.509,Z 301.794,A -85,B 0,C 180,E1 -16607.23,E2 -16607.23} C_VEL
LIN {X 0,Y 443.529,Z 301.794,A -85,B 0,C 180,E1 -16610.828,E2 -16610.828} C_VEL
LIN {X 0,Y 443.539,Z 301.787,A -85,B 0,C 180,E1 -16613.649,E2 -16613.649} C_VEL
LIN {X 0,Y 443.523,Z 301.796,A -85,B 0,C 180,E1 -16616.826,E2 -16616.826} C_VEL
LIN {X 0,Y 443.561,Z 301.903,A -85,B 0,C 180,E1 -16617.114,E2 -16617.114} C_VEL
LIN {X 0,Y 447.073,Z 316.269,A -85,B 0,C 180,E1 -16620.172,E2 -16620.172} C_VEL
LIN {X 0,Y 449.677,Z 328.389,A -85,B 0,C 180,E1 -16622.607,E2 -16622.607} C_VEL
LIN {X 0,Y 450.538,Z 332.731,A -85,B 0,C 180,E1 -16623.453,E2 -16623.453} C_VEL
LIN {X 0,Y 449.57,Z 342.339,A -85,B 0,C 180,E1 -16625.126,E2 -16625.126} C_VEL
LIN {X 0,Y 448.193,Z 353.598,A -85,B 0,C 180,E1 -16627.041,E2 -16627.041} C_VEL
LIN {X 0,Y 453.276,Z 381.005,A -85,B 0,C 180,E1 -16627.836,E2 -16627.836} C_VEL
LIN {X 0,Y 456.376,Z 402.47,A -85,B 0,C 180,E1 -16628.389,E2 -16628.389} C_VEL
LIN {X 0,Y 454.538,Z 491.904,A -85,B 0,C 180,E1 -16629.833,E2 -16629.833} C_VEL
LIN {X 0,Y 453.647,Z 506.705,A -85,B 0,C 180,E1 -16630.242,E2 -16630.242} C_VEL
LIN {X 0,Y 452.457,Z 520.345,A -85,B 0,C 180,E1 -16630.793,E2 -16630.793} C_VEL
LIN {X 0,Y 451.239,Z 532.838,A -85,B 0,C 180,E1 -16631.47,E2 -16631.47} C_VEL
LIN {X 0,Y 449.845,Z 545.257,A -85,B 0,C 180,E1 -16632.327,E2 -16632.327} C_VEL
LIN {X 0,Y 448.228,Z 558.046,A -85,B 0,C 180,E1 -16633.432,E2 -16633.432} C_VEL
LIN {X 0,Y 446.699,Z 568.529,A -85,B 0,C 180,E1 -16634.542,E2 -16634.542} C_VEL
LIN {X 0,Y 445.295,Z 578.979,A -85,B 0,C 180,E1 -16635.891,E2 -16635.891} C_VEL
LIN {X 0,Y 444.184,Z 587.637,A -85,B 0,C 180,E1 -16637.248,E2 -16637.248} C_VEL
LIN {X 0,Y 443.164,Z 595.938,A -85,B 0,C 180,E1 -16638.828,E2 -16638.828} C_VEL
LIN {X 0,Y 442.357,Z 602.734,A -85,B 0,C 180,E1 -16640.432,E2 -16640.432} C_VEL
LIN {X 0,Y 441.74,Z 608.768,A -85,B 0,C 180,E1 -16642.256,E2 -16642.256} C_VEL
LIN {X 0,Y 441.615,Z 613.501,A -85,B 0,C 180,E1 -16644.085,E2 -16644.085} C_VEL
LIN {X 0,Y 441.53,Z 617.665,A -85,B 0,C 180,E1 -16645.453,E2 -16645.453} C_VEL
LIN {X 0,Y 441.51,Z 619.93,A -85,B 0,C 180,E1 -16646.364,E2 -16646.364} C_VEL
LIN {X 0,Y 441.521,Z 621.776,A -85,B 0,C 180,E1 -16647.274,E2 -16647.274} C_VEL
LIN {X 0,Y 441.534,Z 624.288,A -85,B 0,C 180,E1 -16649.093,E2 -16649.093} C_VEL
LIN {X 0,Y 441.513,Z 625.324,A -85,B 0,C 180,E1 -16650.911,E2 -16650.911} C_VEL
LIN {X 0,Y 441.461,Z 624.904,A -85,B 0,C 180,E1 -16652.73,E2 -16652.73} C_VEL
LIN {X 0,Y 441.53,Z 623.046,A -85,B 0,C 180,E1 -16654.552,E2 -16654.552} C_VEL
LIN {X 0,Y 441.707,Z 619.722,A -85,B 0,C 180,E1 -16656.375,E2 -16656.375} C_VEL
LIN {X 0,Y 442.011,Z 616.168,A -85,B 0,C 180,E1 -16657.743,E2 -16657.743} C_VEL
LIN {X 0,Y 442.443,Z 611.717,A -85,B 0,C 180,E1 -16659.111,E2 -16659.111} C_VEL
LIN {X 0,Y 443.378,Z 605.214,A -85,B 0,C 180,E1 -16660.7,E2 -16660.7} C_VEL
LIN {X 0,Y 444.198,Z 598.014,A -85,B 0,C 180,E1 -16662.133,E2 -16662.133} C_VEL
LIN {X 0,Y 445.417,Z 588.737,A -85,B 0,C 180,E1 -16663.646,E2 -16663.646} C_VEL
LIN {X 0,Y 446.811,Z 578.637,A -85,B 0,C 180,E1 -16664.993,E2 -16664.993} C_VEL
LIN {X 0,Y 448.269,Z 567.455,A -85,B 0,C 180,E1 -16666.221,E2 -16666.221} C_VEL
LIN {X 0,Y 449.757,Z 555.08,A -85,B 0,C 180,E1 -16667.33,E2 -16667.33} C_VEL
LIN {X 0,Y 451.376,Z 541.281,A -85,B 0,C 180,E1 -16668.317,E2 -16668.317} C_VEL
LIN {X 0,Y 452.646,Z 528.246,A -85,B 0,C 180,E1 -16669.053,E2 -16669.053} C_VEL
LIN {X 0,Y 453.942,Z 513.518,A -85,B 0,C 180,E1 -16669.679,E2 -16669.679} C_VEL
LIN {X 0,Y 454.933,Z 498.928,A -85,B 0,C 180,E1 -16670.109,E2 -16670.109} C_VEL
LIN {X 0,Y 459.134,Z 403.606,A -85,B 0,C 180,E1 -16672.232,E2 -16672.232} C_VEL
LIN {X 0,Y 457.896,Z 388.46,A -85,B 0,C 180,E1 -16672.738,E2 -16672.738} C_VEL
LIN {X 0,Y 455.226,Z 368.019,A -85,B 0,C 180,E1 -16673.53,E2 -16673.53} C_VEL
LIN {X 0,Y 452.68,Z 353.312,A -85,B 0,C 180,E1 -16674.21,E2 -16674.21} C_VEL
LIN {X 0,Y 451.044,Z 334.396,A -85,B 0,C 180,E1 -16675.621,E2 -16675.621} C_VEL
LIN {X 0,Y 450.14,Z 327.559,A -85,B 0,C 180,E1 -16676.211,E2 -16676.211} C_VEL
LIN {X 0,Y 447.546,Z 318.509,A -85,B 0,C 180,E1 -16677.203,E2 -16677.203} C_VEL
LIN {X 0,Y 445.203,Z 309.84,A -85,B 0,C 180,E1 -16678.23,E2 -16678.23} C_VEL
LIN {X 0,Y 443.524,Z 301.793,A -85,B 0,C 180,E1 -16679.757,E2 -16679.757} C_VEL
LIN {X 0,Y 443.447,Z 301.803,A -85,B 0,C 180,E1 -16683.159,E2 -16683.159} C_VEL
LIN {X 0,Y 443.461,Z 301.804,A -85,B 0,C 180,E1 -16686.337,E2 -16686.337} C_VEL
LIN {X 0,Y 443.467,Z 301.803,A -85,B 0,C 180,E1 -16689.291,E2 -16689.291} C_VEL
LIN {X 0,Y 443.49,Z 301.797,A -85,B 0,C 180,E1 -16692.778,E2 -16692.778} C_VEL
LIN {X 0,Y 443.502,Z 301.797,A -85,B 0,C 180,E1 -16695.98,E2 -16695.98} C_VEL
LIN {X 0,Y 443.478,Z 301.802,A -85,B 0,C 180,E1 -16699.302,E2 -16699.302} C_VEL
LIN {X 0,Y 443.493,Z 301.8,A -85,B 0,C 180,E1 -16702.159,E2 -16702.159} C_VEL
LIN {X 0,Y 443.52,Z 301.796,A -85,B 0,C 180,E1 -16705.351,E2 -16705.351} C_VEL
LIN {X 0,Y 443.504,Z 301.798,A -85,B 0,C 180,E1 -16708.588,E2 -16708.588} C_VEL
LIN {X 0,Y 443.529,Z 301.794,A -85,B 0,C 180,E1 -16711.72,E2 -16711.72} C_VEL
LIN {X 0,Y 443.494,Z 301.802,A -85,B 0,C 180,E1 -16714.759,E2 -16714.759} C_VEL
LIN {X 0,Y 443.52,Z 301.805,A -85,B 0,C 180,E1 -16717.726,E2 -16717.726} C_VEL
LIN {X 0,Y 443.587,Z 301.801,A -85,B 0,C 180,E1 -16719.129,E2 -16719.129} C_VEL
LIN {X 0,Y 448.065,Z 314.648,A -85,B 0,C 180,E1 -16722.044,E2 -16722.044} C_VEL
LIN {X 0,Y 451.459,Z 326.454,A -85,B 0,C 180,E1 -16724.473,E2 -16724.473} C_VEL
LIN {X 0,Y 453.766,Z 337.814,A -85,B 0,C 180,E1 -16726.612,E2 -16726.612} C_VEL
LIN {X 0,Y 453.574,Z 343.383,A -85,B 0,C 180,E1 -16727.514,E2 -16727.514} C_VEL
LIN {X 0,Y 453.346,Z 346.221,A -85,B 0,C 180,E1 -16727.932,E2 -16727.932} C_VEL
LIN {X 0,Y 457.244,Z 362.706,A -85,B 0,C 180,E1 -16728.748,E2 -16728.748} C_VEL
LIN {X 0,Y 460.412,Z 379.837,A -85,B 0,C 180,E1 -16729.481,E2 -16729.481} C_VEL
LIN {X 0,Y 455.526,Z 487.391,A -85,B 0,C 180,E1 -16731.878,E2 -16731.878} C_VEL
LIN {X 0,Y 454.612,Z 501.307,A -85,B 0,C 180,E1 -16732.363,E2 -16732.363} C_VEL
LIN {X 0,Y 453.463,Z 515.012,A -85,B 0,C 180,E1 -16733.013,E2 -16733.013} C_VEL
LIN {X 0,Y 452.144,Z 527.601,A -85,B 0,C 180,E1 -16733.774,E2 -16733.774} C_VEL
LIN {X 0,Y 450.652,Z 540.489,A -85,B 0,C 180,E1 -16734.747,E2 -16734.747} C_VEL
LIN {X 0,Y 449.218,Z 552.406,A -85,B 0,C 180,E1 -16735.864,E2 -16735.864} C_VEL
LIN {X 0,Y 447.842,Z 563.061,A -85,B 0,C 180,E1 -16737.086,E2 -16737.086} C_VEL
LIN {X 0,Y 446.405,Z 572.794,A -85,B 0,C 180,E1 -16738.426,E2 -16738.426} C_VEL
LIN {X 0,Y 445.064,Z 580.94,A -85,B 0,C 180,E1 -16739.775,E2 -16739.775} C_VEL
LIN {X 0,Y 443.944,Z 588.695,A -85,B 0,C 180,E1 -16741.356,E2 -16741.356} C_VEL
LIN {X 0,Y 443.145,Z 594.137,A -85,B 0,C 180,E1 -16742.718,E2 -16742.718} C_VEL
LIN {X 0,Y 442.522,Z 599.81,A -85,B 0,C 180,E1 -16744.539,E2 -16744.539} C_VEL
LIN {X 0,Y 441.958,Z 603.917,A -85,B 0,C 180,E1 -16746.37,E2 -16746.37} C_VEL
LIN {X 0,Y 441.55,Z 606.506,A -85,B 0,C 180,E1 -16748.208,E2 -16748.208} C_VEL
LIN {X 0,Y 441.439,Z 607.609,A -85,B 0,C 180,E1 -16750.052,E2 -16750.052} C_VEL
LIN {X 0,Y 441.257,Z 607.257,A -85,B 0,C 180,E1 -16751.909,E2 -16751.909} C_VEL
LIN {X 0,Y 441.321,Z 605.415,A -85,B 0,C 180,E1 -16753.773,E2 -16753.773} C_VEL
LIN {X 0,Y 441.38,Z 603.92,A -85,B 0,C 180,E1 -16754.709,E2 -16754.709} C_VEL
LIN {X 0,Y 441.462,Z 600.866,A -85,B 0,C 180,E1 -16756.121,E2 -16756.121} C_VEL
LIN {X 0,Y 441.648,Z 596.845,A -85,B 0,C 180,E1 -16757.538,E2 -16757.538} C_VEL
LIN {X 0,Y 441.839,Z 591.732,A -85,B 0,C 180,E1 -16758.965,E2 -16758.965} C_VEL
LIN {X 0,Y 442.261,Z 584.196,A -85,B 0,C 180,E1 -16760.637,E2 -16760.637} C_VEL
LIN {X 0,Y 442.716,Z 576.217,A -85,B 0,C 180,E1 -16762.071,E2 -16762.071} C_VEL
LIN {X 0,Y 443.394,Z 565.737,A -85,B 0,C 180,E1 -16763.613,E2 -16763.613} C_VEL
LIN {X 0,Y 444.093,Z 554.464,A -85,B 0,C 180,E1 -16764.955,E2 -16764.955} C_VEL
LIN {X 0,Y 444.912,Z 542.14,A -85,B 0,C 180,E1 -16766.156,E2 -16766.156} C_VEL
LIN {X 0,Y 445.649,Z 530.06,A -85,B 0,C 180,E1 -16767.117,E2 -16767.117} C_VEL
LIN {X 0,Y 446.348,Z 516.944,A -85,B 0,C 180,E1 -16767.958,E2 -16767.958} C_VEL
LIN {X 0,Y 447.072,Z 502.449,A -85,B 0,C 180,E1 -16768.67,E2 -16768.67} C_VEL
LIN {X 0,Y 447.731,Z 487.475,A -85,B 0,C 180,E1 -16769.203,E2 -16769.203} C_VEL
LIN {X 0,Y 448.141,Z 470.609,A -85,B 0,C 180,E1 -16769.591,E2 -16769.591} C_VEL
LIN {X 0,Y 450.341,Z 374.542,A -85,B 0,C 180,E1 -16771.509,E2 -16771.509} C_VEL
LIN {X 0,Y 446.354,Z 344.063,A -85,B 0,C 180,E1 -16772.287,E2 -16772.287} C_VEL
LIN {X 0,Y 447.432,Z 322.624,A -85,B 0,C 180,E1 -16775.504,E2 -16775.504} C_VEL
LIN {X 0,Y 446.104,Z 314.501,A -85,B 0,C 180,E1 -16776.794,E2 -16776.794} C_VEL
LIN {X 0,Y 443.517,Z 301.797,A -85,B 0,C 180,E1 -16778.87,E2 -16778.87} C_VEL
LIN {X 0,Y 443.505,Z 301.797,A -85,B 0,C 180,E1 -16782.071,E2 -16782.071} C_VEL
LIN {X 0,Y 443.494,Z 301.795,A -85,B 0,C 180,E1 -16785.294,E2 -16785.294} C_VEL
LIN {X 0,Y 443.487,Z 301.801,A -85,B 0,C 180,E1 -16788.442,E2 -16788.442} C_VEL
LIN {X 0,Y 443.47,Z 301.802,A -85,B 0,C 180,E1 -16791.974,E2 -16791.974} C_VEL
LIN {X 0,Y 443.5,Z 301.794,A -85,B 0,C 180,E1 -16795.348,E2 -16795.348} C_VEL
LIN {X 0,Y 443.502,Z 301.796,A -85,B 0,C 180,E1 -16798.586,E2 -16798.586} C_VEL
LIN {X 0,Y 443.499,Z 301.797,A -85,B 0,C 180,E1 -16801.716,E2 -16801.716} C_VEL
LIN {X 0,Y 443.485,Z 301.796,A -85,B 0,C 180,E1 -16804.756,E2 -16804.756} C_VEL
LIN {X 0,Y 443.516,Z 301.796,A -85,B 0,C 180,E1 -16807.724,E2 -16807.724} C_VEL
LIN {X 0,Y 443.565,Z 301.787,A -85,B 0,C 180,E1 -16810.631,E2 -16810.631} C_VEL
LIN {X 0,Y 443.653,Z 301.777,A -85,B 0,C 180,E1 -16814.382,E2 -16814.382} C_VEL
LIN {X 0,Y 443.689,Z 301.774,A -85,B 0,C 180,E1 -16818.177,E2 -16818.177} C_VEL
LIN {X 0,Y 443.688,Z 301.902,A -85,B 0,C 180,E1 -16820.342,E2 -16820.342} C_VEL
LIN {X 0,Y 444.688,Z 307.067,A -85,B 0,C 180,E1 -16821.477,E2 -16821.477} C_VEL
LIN {X 0,Y 449.632,Z 323.181,A -85,B 0,C 180,E1 -16821.938,E2 -16821.938} C_VEL
LIN {X 0,Y 451.549,Z 333.458,A -85,B 0,C 180,E1 -16822.181,E2 -16822.181} C_VEL
LIN {X 0,Y 449.664,Z 441.922,A -85,B 0,C 180,E1 -16823.906,E2 -16823.906} C_VEL
LIN {X 0,Y 449.249,Z 456.578,A -85,B 0,C 180,E1 -16824.322,E2 -16824.322} C_VEL
LIN {X 0,Y 448.709,Z 470.485,A -85,B 0,C 180,E1 -16824.904,E2 -16824.904} C_VEL
LIN {X 0,Y 448.007,Z 483.426,A -85,B 0,C 180,E1 -16825.627,E2 -16825.627} C_VEL
LIN {X 0,Y 447.232,Z 495.957,A -85,B 0,C 180,E1 -16826.518,E2 -16826.518} C_VEL
LIN {X 0,Y 446.152,Z 507.462,A -85,B 0,C 180,E1 -16827.523,E2 -16827.523} C_VEL
LIN {X 0,Y 445.473,Z 517.927,A -85,B 0,C 180,E1 -16828.646,E2 -16828.646} C_VEL
LIN {X 0,Y 444.478,Z 528.386,A -85,B 0,C 180,E1 -16829.998,E2 -16829.998} C_VEL
LIN {X 0,Y 443.747,Z 537.006,A -85,B 0,C 180,E1 -16831.355,E2 -16831.355} C_VEL
LIN {X 0,Y 443.042,Z 544.197,A -85,B 0,C 180,E1 -16832.716,E2 -16832.716} C_VEL
LIN {X 0,Y 442.735,Z 550.652,A -85,B 0,C 180,E1 -16834.207,E2 -16834.207} C_VEL
LIN {X 0,Y 442.282,Z 556.535,A -85,B 0,C 180,E1 -16835.906,E2 -16835.906} C_VEL
LIN {X 0,Y 441.911,Z 561.307,A -85,B 0,C 180,E1 -16837.741,E2 -16837.741} C_VEL
LIN {X 0,Y 441.782,Z 563.862,A -85,B 0,C 180,E1 -16839.12,E2 -16839.12} C_VEL
LIN {X 0,Y 441.703,Z 566.092,A -85,B 0,C 180,E1 -16840.967,E2 -16840.967} C_VEL
LIN {X 0,Y 441.691,Z 566.233,A -85,B 0,C 180,E1 -16841.182,E2 -16841.182} C_VEL
LIN {X 0,Y 441.024,Z 566.771,A -85,B 0,C 180,E1 -16841.942,E2 -16841.942} C_VEL
LIN {X 0,Y 438.244,Z 567.202,A -85,B 0,C 180,E1 -16843.181,E2 -16843.181} C_VEL
LIN {X 0,Y 435.936,Z 567.165,A -85,B 0,C 180,E1 -16844.18,E2 -16844.18} C_VEL
LIN {X 0,Y 434.988,Z 566.813,A -85,B 0,C 180,E1 -16844.949,E2 -16844.949} C_VEL
LIN {X 0,Y 434.933,Z 566.595,A -85,B 0,C 180,E1 -16845.208,E2 -16845.208} C_VEL
LIN {X 0,Y 435.206,Z 564.852,A -85,B 0,C 180,E1 -16846.837,E2 -16846.837} C_VEL
LIN {X 0,Y 435.803,Z 561.414,A -85,B 0,C 180,E1 -16848.748,E2 -16848.748} C_VEL
LIN {X 0,Y 436.66,Z 556.402,A -85,B 0,C 180,E1 -16850.662,E2 -16850.662} C_VEL
LIN {X 0,Y 437.431,Z 551.494,A -85,B 0,C 180,E1 -16852.101,E2 -16852.101} C_VEL
LIN {X 0,Y 438.626,Z 544.339,A -85,B 0,C 180,E1 -16853.777,E2 -16853.777} C_VEL
LIN {X 0,Y 439.855,Z 536.738,A -85,B 0,C 180,E1 -16855.217,E2 -16855.217} C_VEL
LIN {X 0,Y 441.249,Z 527.609,A -85,B 0,C 180,E1 -16856.641,E2 -16856.641} C_VEL
LIN {X 0,Y 442.676,Z 517.682,A -85,B 0,C 180,E1 -16857.916,E2 -16857.916} C_VEL
LIN {X 0,Y 444.054,Z 507.348,A -85,B 0,C 180,E1 -16859.012,E2 -16859.012} C_VEL
LIN {X 0,Y 445.381,Z 495.981,A -85,B 0,C 180,E1 -16860.008,E2 -16860.008} C_VEL
LIN {X 0,Y 446.619,Z 483.33,A -85,B 0,C 180,E1 -16860.903,E2 -16860.903} C_VEL
LIN {X 0,Y 447.542,Z 470.483,A -85,B 0,C 180,E1 -16861.618,E2 -16861.618} C_VEL
LIN {X 0,Y 448.446,Z 456.173,A -85,B 0,C 180,E1 -16862.203,E2 -16862.203} C_VEL
LIN {X 0,Y 448.95,Z 441.893,A -85,B 0,C 180,E1 -16862.595,E2 -16862.595} C_VEL
LIN {X 0,Y 451.099,Z 339.329,A -85,B 0,C 180,E1 -16864.271,E2 -16864.271} C_VEL
LIN {X 0,Y 445.007,Z 324.466,A -85,B 0,C 180,E1 -16864.928,E2 -16864.928} C_VEL
LIN {X 0,Y 437.735,Z 308.445,A -85,B 0,C 180,E1 -16865.731,E2 -16865.731} C_VEL
LIN {X 0,Y 436.411,Z 302.682,A -85,B 0,C 180,E1 -16867.268,E2 -16867.268} C_VEL
LIN {X 0,Y 436.402,Z 302.686,A -85,B 0,C 180,E1 -16869.939,E2 -16869.939} C_VEL
LIN {X 0,Y 436.427,Z 302.677,A -85,B 0,C 180,E1 -16872.415,E2 -16872.415} C_VEL
LIN {X 0,Y 436.426,Z 302.664,A -85,B 0,C 180,E1 -16875.075,E2 -16875.075} C_VEL
LIN {X 0,Y 436.426,Z 302.679,A -85,B 0,C 180,E1 -16877.617,E2 -16877.617} C_VEL
LIN {X 0,Y 436.419,Z 302.678,A -85,B 0,C 180,E1 -16880.384,E2 -16880.384} C_VEL
LIN {X 0,Y 436.428,Z 302.658,A -85,B 0,C 180,E1 -16883.571,E2 -16883.571} C_VEL
LIN {X 0,Y 436.439,Z 302.676,A -85,B 0,C 180,E1 -16886.564,E2 -16886.564} C_VEL
LIN {X 0,Y 436.445,Z 302.67,A -85,B 0,C 180,E1 -16889.099,E2 -16889.099} C_VEL
LIN {X 0,Y 436.476,Z 302.664,A -85,B 0,C 180,E1 -16892.265,E2 -16892.265} C_VEL
LIN {X 0,Y 436.431,Z 302.68,A -85,B 0,C 180,E1 -16895.337,E2 -16895.337} C_VEL
LIN {X 0,Y 436.464,Z 302.673,A -85,B 0,C 180,E1 -16898.339,E2 -16898.339} C_VEL
LIN {X 0,Y 436.508,Z 302.659,A -85,B 0,C 180,E1 -16901.281,E2 -16901.281} C_VEL
LIN {X 0,Y 436.542,Z 302.658,A -85,B 0,C 180,E1 -16905.124,E2 -16905.124} C_VEL
LIN {X 0,Y 436.615,Z 302.654,A -85,B 0,C 180,E1 -16908.11,E2 -16908.11} C_VEL
LIN {X 0,Y 436.668,Z 302.64,A -85,B 0,C 180,E1 -16911.699,E2 -16911.699} C_VEL
LIN {X 0,Y 436.701,Z 302.643,A -85,B 0,C 180,E1 -16914.478,E2 -16914.478} C_VEL
LIN {X 0,Y 436.729,Z 302.625,A -85,B 0,C 180,E1 -16916.322,E2 -16916.322} C_VEL
LIN {X 0,Y 436.758,Z 302.634,A -85,B 0,C 180,E1 -16920,E2 -16920} C_VEL
LIN {X 0,Y 436.732,Z 302.639,A -85,B 0,C 180,E1 -16923.678,E2 -16923.678} C_VEL
LIN {X 0,Y 436.711,Z 302.636,A -85,B 0,C 180,E1 -16926.446,E2 -16926.446} C_VEL
LIN {X 0,Y 436.613,Z 302.655,A -85,B 0,C 180,E1 -16929.232,E2 -16929.232} C_VEL
